// TwinCAT 3 PLC project MoXX_2TilesDemo
// ProgramVersion: 3.1.4026.13
// libraries:
//   Tc2_EtherCAT, * (Beckhoff Automation GmbH)
//   Tc2_MC2, * (Beckhoff Automation GmbH)
//   Tc2_MC2_Camming, * (Beckhoff Automation GmbH)
//   Tc2_NCI, * (Beckhoff Automation GmbH)
//   Tc2_Standard, * (Beckhoff Automation GmbH)
//   Tc2_System, * (Beckhoff Automation GmbH)
//   Tc2_Utilities, * (Beckhoff Automation GmbH)
//   Tc3_Mc3PlanarMotion, * (Beckhoff Automation GmbH)
//   Tc3_Module, * (Beckhoff Automation GmbH)
//   Tc3_Physics, * (Beckhoff Automation GmbH)
//   Tc3_XPlanarStandard, * (Beckhoff Automation GmbH)
//   Tc3_XPlanarUtility, * (Beckhoff Automation GmbH)
// project tree:
//   GVLs/ GVL10_VAR_PRG.TcGVL
//   / PlcTask.TcTTO
//   POUs/10_GeneralPlcBlocks/ Blinker.TcPOU, ClockGenerator.TcPOU, GeneralPlc.TcPOU
//   POUs/10_GeneralPlcBlocks/Components/ FB_Blinker.TcPOU, F_Scaling.TcPOU
//   POUs/CustomerTemplates/GCode/ FB_GCode.TcPOU, I_GCode.TcIO
//   POUs/CustomerTemplates/SwivelMovement/ FB_SwivelMovement.TcPOU, I_SwivelMovement.TcIO
//   POUs/CustomerTemplates/Shake/ FB_ShakeMovement.TcPOU, I_ShakeMovement.TcIO
//   POUs/ FB_MoverApplication.TcPOU, FB_WriteLog.TcPOU, I_MoverApplication.TcIO, MAIN.TcPOU
// real-time tasks:
//   TASK Job Task: cycle default, priority 32
//   TASK MC-Task (MET): cycle T#2ms, priority 3, ADS port 521
//   TASK MC-Task (MPT): cycle T#10ms, priority 8, ADS port 531
//   TASK PlcTask: cycle T#10ms, priority 6, ADS port 352
//   TASK XPlanar Task3: cycle T#250us, priority 1, ADS port 350
// motion (NC):
//   TASK NC-Task 1 SAF: cycle T#2ms, priority 4, ADS port 501
//   TASK NC-Task 1 SVB: cycle T#10ms, priority 9, ADS port 511
//   AXIS MasterShake (id 7)
//     General: UnitFlags=#x00000004
//     OtherSettings: AllowMotionCmdToSlave=true
//     encoder EncType=1
//     drive DrvType=5
//       Analog: TorqueSetpointScale=10, ScaleFactorActTorque=0.1
//       TimeComp: TaskDelayCycles=1
//     controller CtrType=1
//       CtrPara: PriorControlFactor=1
//         Observer: BandWidth=20
//   AXIS Axis a (id 8)
//     OtherSettings: AllowMotionCmdToSlave=true
//     encoder EncType=1
//     drive DrvType=5
//       Analog: TorqueSetpointScale=10, ScaleFactorActTorque=0.1
//       TimeComp: TaskDelayCycles=1
//     controller CtrType=1
//       CtrPara: PriorControlFactor=1
//         Observer: BandWidth=20
//   AXIS Axis b (id 9)
//     OtherSettings: AllowMotionCmdToSlave=true
//     encoder EncType=1
//     drive DrvType=5
//       Analog: TorqueSetpointScale=10, ScaleFactorActTorque=0.1
//       TimeComp: TaskDelayCycles=1
//     controller CtrType=1
//       CtrPara: PriorControlFactor=1
//         Observer: BandWidth=20
//   AXIS Axis x (id 10)
//     OtherSettings: AllowMotionCmdToSlave=true
//     encoder EncType=1
//     drive DrvType=5
//       Analog: TorqueSetpointScale=10, ScaleFactorActTorque=0.1
//       TimeComp: TaskDelayCycles=1
//     controller CtrType=1
//       CtrPara: PriorControlFactor=1
//         Observer: BandWidth=20
//   AXIS Axis y (id 11)
//     OtherSettings: AllowMotionCmdToSlave=true
//     encoder EncType=1
//     drive DrvType=5
//       Analog: TorqueSetpointScale=10, ScaleFactorActTorque=0.1
//       TimeComp: TaskDelayCycles=1
//     controller CtrType=1
//       CtrPara: PriorControlFactor=1
//         Observer: BandWidth=20
//   AXIS Axis 1 (id 1)
//     OtherSettings: AllowMotionCmdToSlave=true
//     encoder EncType=1
//     drive DrvType=5
//       Analog: TorqueSetpointScale=10, ScaleFactorActTorque=0.1
//       TimeComp: TaskDelayCycles=1
//     controller CtrType=1
//       CtrPara: PriorControlFactor=1
//         Observer: BandWidth=20
//   AXIS Axis 2 (id 2)
//     OtherSettings: AllowMotionCmdToSlave=true
//     encoder EncType=1
//     drive DrvType=5
//       Analog: TorqueSetpointScale=10, ScaleFactorActTorque=0.1
//       TimeComp: TaskDelayCycles=1
//     controller CtrType=1
//       CtrPara: PriorControlFactor=1
//         Observer: BandWidth=20
//   AXIS Axis 3 (id 3)
//     OtherSettings: AllowMotionCmdToSlave=true
//     encoder EncType=1
//     drive DrvType=5
//       Analog: TorqueSetpointScale=10, ScaleFactorActTorque=0.1
//       TimeComp: TaskDelayCycles=1
//     controller CtrType=1
//       CtrPara: PriorControlFactor=1
//         Observer: BandWidth=20
//   AXIS Axis 4 (id 4)
//     OtherSettings: AllowMotionCmdToSlave=true
//     encoder EncType=1
//     drive DrvType=5
//       Analog: TorqueSetpointScale=10, ScaleFactorActTorque=0.1
//       TimeComp: TaskDelayCycles=1
//     controller CtrType=1
//       CtrPara: PriorControlFactor=1
//         Observer: BandWidth=20
//   AXIS Axis 5 (id 5)
//     OtherSettings: AllowMotionCmdToSlave=true
//     encoder EncType=1
//     drive DrvType=5
//       Analog: TorqueSetpointScale=10, ScaleFactorActTorque=0.1
//       TimeComp: TaskDelayCycles=1
//     controller CtrType=1
//       CtrPara: PriorControlFactor=1
//         Observer: BandWidth=20
//   AXIS Axis 6 (id 6)
//     OtherSettings: AllowMotionCmdToSlave=true
//     encoder EncType=1
//     drive DrvType=5
//       Analog: TorqueSetpointScale=10, ScaleFactorActTorque=0.1
//       TimeComp: TaskDelayCycles=1
//     controller CtrType=1
//       CtrPara: PriorControlFactor=1
//         Observer: BandWidth=20
// I/O:
//   DEVICE Device 5 (EtherCAT), AmsNetId 5.91.77.10.6.1
//     Term 1 (APS4322-7000) [APS4322-7000 Drive]
//       Term 2 (APS4322-5000) [APS4322-5000 Feedback]
//     Term 3 (APS4322-7000) [APS4322-7000 Drive]
//       Term 4 (APS4322-5000) [APS4322-5000 Feedback]
//   DEVICE Gerät 4 (EtherCAT), AmsNetId 169.254.59.222.5.1
//     Box 5 (EP2316-0003) [EP2316-0003 8 K. Dig. Ein, 10µs, 8 K. Dig. Aus 24V, 0,5A, Diagnose, 10-Pol Steckverbinder]
// variable links:
//   Device 5 (EtherCAT) <-> TcCOM Objects/XPlanar/Part1/Tile1
//     Term 1 (APS4322-7000)/APS Comm Inputs/CommStatusWord <-> Data Pointer/MoverCommStatusWord
//     Term 1 (APS4322-7000)/APS Comm Inputs/Data {1..4} <-> Data Pointer/MoverCommDataIn[{0..3}]  (4 links)
//     Term 1 (APS4322-7000)/APS Comm Outputs/CommControlWord <-> Data Pointer/MoverCommControlWord
//     Term 1 (APS4322-7000)/APS Comm Outputs/Data 1 <-> Data Pointer/MoverCommDataOut
//     Term 1 (APS4322-7000)/APS Diagdata/DC Link Voltage <-> Data Pointer/DcLinkVoltage
//     Term 1 (APS4322-7000)/APS Diagdata/Power supply current <-> Data Pointer/PowerSupplyCurrent
//     Term 1 (APS4322-7000)/APS Inputs/StatusWord <-> Data Pointer/PowerUnitStatusWord
//     Term 1 (APS4322-7000)/APS Outputs/ControlWord <-> Data Pointer/PowerUnitControlWord
//     Term 1 (APS4322-7000)/APS Outputs/Current D 0X0 <-> Data Pointer/DCurrentSetPoints[0]
//     Term 1 (APS4322-7000)/APS Outputs/Current D 0X1 <-> Data Pointer/DCurrentSetPoints[1]
//     Term 1 (APS4322-7000)/APS Outputs/Current D 0X2 <-> Data Pointer/DCurrentSetPoints[2]
//     Term 1 (APS4322-7000)/APS Outputs/Current D 1X0 <-> Data Pointer/DCurrentSetPoints[6]
//     Term 1 (APS4322-7000)/APS Outputs/Current D 1X1 <-> Data Pointer/DCurrentSetPoints[7]
//     Term 1 (APS4322-7000)/APS Outputs/Current D 1X2 <-> Data Pointer/DCurrentSetPoints[8]
//     Term 1 (APS4322-7000)/APS Outputs/Current D 2X0 <-> Data Pointer/DCurrentSetPoints[12]
//     Term 1 (APS4322-7000)/APS Outputs/Current D 2X1 <-> Data Pointer/DCurrentSetPoints[13]
//     Term 1 (APS4322-7000)/APS Outputs/Current D 2X2 <-> Data Pointer/DCurrentSetPoints[14]
//     Term 1 (APS4322-7000)/APS Outputs/Current D 3X0 <-> Data Pointer/DCurrentSetPoints[18]
//     Term 1 (APS4322-7000)/APS Outputs/Current D 3X1 <-> Data Pointer/DCurrentSetPoints[19]
//     Term 1 (APS4322-7000)/APS Outputs/Current D 3X2 <-> Data Pointer/DCurrentSetPoints[20]
//     Term 1 (APS4322-7000)/APS Outputs/Current D 0Y0 <-> Data Pointer/DCurrentSetPoints[3]
//     Term 1 (APS4322-7000)/APS Outputs/Current D 0Y1 <-> Data Pointer/DCurrentSetPoints[4]
//     Term 1 (APS4322-7000)/APS Outputs/Current D 0Y2 <-> Data Pointer/DCurrentSetPoints[5]
//     Term 1 (APS4322-7000)/APS Outputs/Current D 1Y0 <-> Data Pointer/DCurrentSetPoints[9]
//     Term 1 (APS4322-7000)/APS Outputs/Current D 1Y1 <-> Data Pointer/DCurrentSetPoints[10]
//     Term 1 (APS4322-7000)/APS Outputs/Current D 1Y2 <-> Data Pointer/DCurrentSetPoints[11]
//     Term 1 (APS4322-7000)/APS Outputs/Current D 2Y0 <-> Data Pointer/DCurrentSetPoints[15]
//     Term 1 (APS4322-7000)/APS Outputs/Current D 2Y1 <-> Data Pointer/DCurrentSetPoints[16]
//     Term 1 (APS4322-7000)/APS Outputs/Current D 2Y2 <-> Data Pointer/DCurrentSetPoints[17]
//     Term 1 (APS4322-7000)/APS Outputs/Current D 3Y0 <-> Data Pointer/DCurrentSetPoints[21]
//     Term 1 (APS4322-7000)/APS Outputs/Current D 3Y1 <-> Data Pointer/DCurrentSetPoints[22]
//     Term 1 (APS4322-7000)/APS Outputs/Current D 3Y2 <-> Data Pointer/DCurrentSetPoints[23]
//     Term 1 (APS4322-7000)/APS Outputs/Current Q 0X0 <-> Data Pointer/QCurrentSetPoints[0]
//     Term 1 (APS4322-7000)/APS Outputs/Current Q 0X1 <-> Data Pointer/QCurrentSetPoints[1]
//     Term 1 (APS4322-7000)/APS Outputs/Current Q 0X2 <-> Data Pointer/QCurrentSetPoints[2]
//     Term 1 (APS4322-7000)/APS Outputs/Current Q 1X0 <-> Data Pointer/QCurrentSetPoints[6]
//     Term 1 (APS4322-7000)/APS Outputs/Current Q 1X1 <-> Data Pointer/QCurrentSetPoints[7]
//     Term 1 (APS4322-7000)/APS Outputs/Current Q 1X2 <-> Data Pointer/QCurrentSetPoints[8]
//     Term 1 (APS4322-7000)/APS Outputs/Current Q 2X0 <-> Data Pointer/QCurrentSetPoints[12]
//     Term 1 (APS4322-7000)/APS Outputs/Current Q 2X1 <-> Data Pointer/QCurrentSetPoints[13]
//     Term 1 (APS4322-7000)/APS Outputs/Current Q 2X2 <-> Data Pointer/QCurrentSetPoints[14]
//     Term 1 (APS4322-7000)/APS Outputs/Current Q 3X0 <-> Data Pointer/QCurrentSetPoints[18]
//     Term 1 (APS4322-7000)/APS Outputs/Current Q 3X1 <-> Data Pointer/QCurrentSetPoints[19]
//     Term 1 (APS4322-7000)/APS Outputs/Current Q 3X2 <-> Data Pointer/QCurrentSetPoints[20]
//     Term 1 (APS4322-7000)/APS Outputs/Current Q 0Y0 <-> Data Pointer/QCurrentSetPoints[3]
//     Term 1 (APS4322-7000)/APS Outputs/Current Q 0Y1 <-> Data Pointer/QCurrentSetPoints[4]
//     Term 1 (APS4322-7000)/APS Outputs/Current Q 0Y2 <-> Data Pointer/QCurrentSetPoints[5]
//     Term 1 (APS4322-7000)/APS Outputs/Current Q 1Y0 <-> Data Pointer/QCurrentSetPoints[9]
//     Term 1 (APS4322-7000)/APS Outputs/Current Q 1Y1 <-> Data Pointer/QCurrentSetPoints[10]
//     Term 1 (APS4322-7000)/APS Outputs/Current Q 1Y2 <-> Data Pointer/QCurrentSetPoints[11]
//     Term 1 (APS4322-7000)/APS Outputs/Current Q 2Y0 <-> Data Pointer/QCurrentSetPoints[15]
//     Term 1 (APS4322-7000)/APS Outputs/Current Q 2Y1 <-> Data Pointer/QCurrentSetPoints[16]
//     Term 1 (APS4322-7000)/APS Outputs/Current Q 2Y2 <-> Data Pointer/QCurrentSetPoints[17]
//     Term 1 (APS4322-7000)/APS Outputs/Current Q 3Y0 <-> Data Pointer/QCurrentSetPoints[21]
//     Term 1 (APS4322-7000)/APS Outputs/Current Q 3Y1 <-> Data Pointer/QCurrentSetPoints[22]
//     Term 1 (APS4322-7000)/APS Outputs/Current Q 3Y2 <-> Data Pointer/QCurrentSetPoints[23]
//     Term 1 (APS4322-7000)/APS Outputs/PhiE 0X0 <-> Data Pointer/PhiSetPoints[0]
//     Term 1 (APS4322-7000)/APS Outputs/PhiE 0X1 <-> Data Pointer/PhiSetPoints[1]
//     Term 1 (APS4322-7000)/APS Outputs/PhiE 0X2 <-> Data Pointer/PhiSetPoints[2]
//     Term 1 (APS4322-7000)/APS Outputs/PhiE 1X0 <-> Data Pointer/PhiSetPoints[6]
//     Term 1 (APS4322-7000)/APS Outputs/PhiE 1X1 <-> Data Pointer/PhiSetPoints[7]
//     Term 1 (APS4322-7000)/APS Outputs/PhiE 1X2 <-> Data Pointer/PhiSetPoints[8]
//     Term 1 (APS4322-7000)/APS Outputs/PhiE 2X0 <-> Data Pointer/PhiSetPoints[12]
//     Term 1 (APS4322-7000)/APS Outputs/PhiE 2X1 <-> Data Pointer/PhiSetPoints[13]
//     Term 1 (APS4322-7000)/APS Outputs/PhiE 2X2 <-> Data Pointer/PhiSetPoints[14]
//     Term 1 (APS4322-7000)/APS Outputs/PhiE 3X0 <-> Data Pointer/PhiSetPoints[18]
//     Term 1 (APS4322-7000)/APS Outputs/PhiE 3X1 <-> Data Pointer/PhiSetPoints[19]
//     Term 1 (APS4322-7000)/APS Outputs/PhiE 3X2 <-> Data Pointer/PhiSetPoints[20]
//     Term 1 (APS4322-7000)/APS Outputs/PhiE 0Y0 <-> Data Pointer/PhiSetPoints[3]
//     Term 1 (APS4322-7000)/APS Outputs/PhiE 0Y1 <-> Data Pointer/PhiSetPoints[4]
//     Term 1 (APS4322-7000)/APS Outputs/PhiE 0Y2 <-> Data Pointer/PhiSetPoints[5]
//     Term 1 (APS4322-7000)/APS Outputs/PhiE 1Y0 <-> Data Pointer/PhiSetPoints[9]
//     Term 1 (APS4322-7000)/APS Outputs/PhiE 1Y1 <-> Data Pointer/PhiSetPoints[10]
//     Term 1 (APS4322-7000)/APS Outputs/PhiE 1Y2 <-> Data Pointer/PhiSetPoints[11]
//     Term 1 (APS4322-7000)/APS Outputs/PhiE 2Y0 <-> Data Pointer/PhiSetPoints[15]
//     Term 1 (APS4322-7000)/APS Outputs/PhiE 2Y1 <-> Data Pointer/PhiSetPoints[16]
//     Term 1 (APS4322-7000)/APS Outputs/PhiE 2Y2 <-> Data Pointer/PhiSetPoints[17]
//     Term 1 (APS4322-7000)/APS Outputs/PhiE 3Y0 <-> Data Pointer/PhiSetPoints[21]
//     Term 1 (APS4322-7000)/APS Outputs/PhiE 3Y1 <-> Data Pointer/PhiSetPoints[22]
//     Term 1 (APS4322-7000)/APS Outputs/PhiE 3Y2 <-> Data Pointer/PhiSetPoints[23]
//     Term 1 (APS4322-7000)/Term 2 (APS4322-5000)/FB Inputs/A{0..8 step 2} X-Field <-> Data Pointer/HallSensorFieldsXYZ[{0..12 step 3}]  (5 links)
//     Term 1 (APS4322-7000)/Term 2 (APS4322-5000)/FB Inputs/A{0..8 step 2} Y-Field <-> Data Pointer/HallSensorFieldsXYZ[{1..13 step 3}]  (5 links)
//     Term 1 (APS4322-7000)/Term 2 (APS4322-5000)/FB Inputs/A{0..8 step 2} Z-Field <-> Data Pointer/HallSensorFieldsXYZ[{2..14 step 3}]  (5 links)
//     Term 1 (APS4322-7000)/Term 2 (APS4322-5000)/FB Inputs/B{1..9 step 2} X-Field <-> Data Pointer/HallSensorFieldsXYZ[{15..27 step 3}]  (5 links)
//     Term 1 (APS4322-7000)/Term 2 (APS4322-5000)/FB Inputs/B{1..9 step 2} Y-Field <-> Data Pointer/HallSensorFieldsXYZ[{16..28 step 3}]  (5 links)
//     Term 1 (APS4322-7000)/Term 2 (APS4322-5000)/FB Inputs/B{1..9 step 2} Z-Field <-> Data Pointer/HallSensorFieldsXYZ[{17..29 step 3}]  (5 links)
//     Term 1 (APS4322-7000)/Term 2 (APS4322-5000)/FB Inputs/C{0..8 step 2} X-Field <-> Data Pointer/HallSensorFieldsXYZ[{30..42 step 3}]  (5 links)
//     Term 1 (APS4322-7000)/Term 2 (APS4322-5000)/FB Inputs/C{0..8 step 2} Y-Field <-> Data Pointer/HallSensorFieldsXYZ[{31..43 step 3}]  (5 links)
//     Term 1 (APS4322-7000)/Term 2 (APS4322-5000)/FB Inputs/C{0..8 step 2} Z-Field <-> Data Pointer/HallSensorFieldsXYZ[{32..44 step 3}]  (5 links)
//     Term 1 (APS4322-7000)/Term 2 (APS4322-5000)/FB Inputs/D{1..9 step 2} X-Field <-> Data Pointer/HallSensorFieldsXYZ[{45..57 step 3}]  (5 links)
//     Term 1 (APS4322-7000)/Term 2 (APS4322-5000)/FB Inputs/D{1..9 step 2} Y-Field <-> Data Pointer/HallSensorFieldsXYZ[{46..58 step 3}]  (5 links)
//     Term 1 (APS4322-7000)/Term 2 (APS4322-5000)/FB Inputs/D{1..9 step 2} Z-Field <-> Data Pointer/HallSensorFieldsXYZ[{47..59 step 3}]  (5 links)
//     Term 1 (APS4322-7000)/Term 2 (APS4322-5000)/FB Inputs/E{0..8 step 2} X-Field <-> Data Pointer/HallSensorFieldsXYZ[{60..72 step 3}]  (5 links)
//     Term 1 (APS4322-7000)/Term 2 (APS4322-5000)/FB Inputs/E{0..8 step 2} Y-Field <-> Data Pointer/HallSensorFieldsXYZ[{61..73 step 3}]  (5 links)
//     Term 1 (APS4322-7000)/Term 2 (APS4322-5000)/FB Inputs/E{0..8 step 2} Z-Field <-> Data Pointer/HallSensorFieldsXYZ[{62..74 step 3}]  (5 links)
//     Term 1 (APS4322-7000)/Term 2 (APS4322-5000)/FB Inputs/F{1..9 step 2} X-Field <-> Data Pointer/HallSensorFieldsXYZ[{75..87 step 3}]  (5 links)
//     Term 1 (APS4322-7000)/Term 2 (APS4322-5000)/FB Inputs/F{1..9 step 2} Y-Field <-> Data Pointer/HallSensorFieldsXYZ[{76..88 step 3}]  (5 links)
//     Term 1 (APS4322-7000)/Term 2 (APS4322-5000)/FB Inputs/F{1..9 step 2} Z-Field <-> Data Pointer/HallSensorFieldsXYZ[{77..89 step 3}]  (5 links)
//     Term 1 (APS4322-7000)/Term 2 (APS4322-5000)/FB Inputs/G{0..8 step 2} X-Field <-> Data Pointer/HallSensorFieldsXYZ[{90..102 step 3}]  (5 links)
//     Term 1 (APS4322-7000)/Term 2 (APS4322-5000)/FB Inputs/G{0..8 step 2} Y-Field <-> Data Pointer/HallSensorFieldsXYZ[{91..103 step 3}]  (5 links)
//     Term 1 (APS4322-7000)/Term 2 (APS4322-5000)/FB Inputs/G{0..8 step 2} Z-Field <-> Data Pointer/HallSensorFieldsXYZ[{92..104 step 3}]  (5 links)
//     Term 1 (APS4322-7000)/Term 2 (APS4322-5000)/FB Inputs/H{1..9 step 2} X-Field <-> Data Pointer/HallSensorFieldsXYZ[{105..117 step 3}]  (5 links)
//     Term 1 (APS4322-7000)/Term 2 (APS4322-5000)/FB Inputs/H{1..9 step 2} Y-Field <-> Data Pointer/HallSensorFieldsXYZ[{106..118 step 3}]  (5 links)
//     Term 1 (APS4322-7000)/Term 2 (APS4322-5000)/FB Inputs/H{1..9 step 2} Z-Field <-> Data Pointer/HallSensorFieldsXYZ[{107..119 step 3}]  (5 links)
//     Term 1 (APS4322-7000)/Term 2 (APS4322-5000)/FB Inputs/I{0..8 step 2} X-Field <-> Data Pointer/HallSensorFieldsXYZ[{120..132 step 3}]  (5 links)
//     Term 1 (APS4322-7000)/Term 2 (APS4322-5000)/FB Inputs/I{0..8 step 2} Y-Field <-> Data Pointer/HallSensorFieldsXYZ[{121..133 step 3}]  (5 links)
//     Term 1 (APS4322-7000)/Term 2 (APS4322-5000)/FB Inputs/I{0..8 step 2} Z-Field <-> Data Pointer/HallSensorFieldsXYZ[{122..134 step 3}]  (5 links)
//     Term 1 (APS4322-7000)/Term 2 (APS4322-5000)/FB Inputs/J{1..9 step 2} X-Field <-> Data Pointer/HallSensorFieldsXYZ[{135..147 step 3}]  (5 links)
//     Term 1 (APS4322-7000)/Term 2 (APS4322-5000)/FB Inputs/J{1..9 step 2} Y-Field <-> Data Pointer/HallSensorFieldsXYZ[{136..148 step 3}]  (5 links)
//     Term 1 (APS4322-7000)/Term 2 (APS4322-5000)/FB Inputs/J{1..9 step 2} Z-Field <-> Data Pointer/HallSensorFieldsXYZ[{137..149 step 3}]  (5 links)
//     Term 1 (APS4322-7000)/Term 2 (APS4322-5000)/FB Inputs/Status <-> Data Pointer/FeedbackStatus
//   Device 5 (EtherCAT) <-> TcCOM Objects/XPlanar/Part1/Tile2
//     Term 3 (APS4322-7000)/APS Comm Inputs/CommStatusWord <-> Data Pointer/MoverCommStatusWord
//     Term 3 (APS4322-7000)/APS Comm Inputs/Data {1..4} <-> Data Pointer/MoverCommDataIn[{0..3}]  (4 links)
//     Term 3 (APS4322-7000)/APS Comm Outputs/CommControlWord <-> Data Pointer/MoverCommControlWord
//     Term 3 (APS4322-7000)/APS Comm Outputs/Data 1 <-> Data Pointer/MoverCommDataOut
//     Term 3 (APS4322-7000)/APS Diagdata/DC Link Voltage <-> Data Pointer/DcLinkVoltage
//     Term 3 (APS4322-7000)/APS Diagdata/Power supply current <-> Data Pointer/PowerSupplyCurrent
//     Term 3 (APS4322-7000)/APS Inputs/StatusWord <-> Data Pointer/PowerUnitStatusWord
//     Term 3 (APS4322-7000)/APS Outputs/ControlWord <-> Data Pointer/PowerUnitControlWord
//     Term 3 (APS4322-7000)/APS Outputs/Current D 0X0 <-> Data Pointer/DCurrentSetPoints[0]
//     Term 3 (APS4322-7000)/APS Outputs/Current D 0X1 <-> Data Pointer/DCurrentSetPoints[1]
//     Term 3 (APS4322-7000)/APS Outputs/Current D 0X2 <-> Data Pointer/DCurrentSetPoints[2]
//     Term 3 (APS4322-7000)/APS Outputs/Current D 1X0 <-> Data Pointer/DCurrentSetPoints[6]
//     Term 3 (APS4322-7000)/APS Outputs/Current D 1X1 <-> Data Pointer/DCurrentSetPoints[7]
//     Term 3 (APS4322-7000)/APS Outputs/Current D 1X2 <-> Data Pointer/DCurrentSetPoints[8]
//     Term 3 (APS4322-7000)/APS Outputs/Current D 2X0 <-> Data Pointer/DCurrentSetPoints[12]
//     Term 3 (APS4322-7000)/APS Outputs/Current D 2X1 <-> Data Pointer/DCurrentSetPoints[13]
//     Term 3 (APS4322-7000)/APS Outputs/Current D 2X2 <-> Data Pointer/DCurrentSetPoints[14]
//     Term 3 (APS4322-7000)/APS Outputs/Current D 3X0 <-> Data Pointer/DCurrentSetPoints[18]
//     Term 3 (APS4322-7000)/APS Outputs/Current D 3X1 <-> Data Pointer/DCurrentSetPoints[19]
//     Term 3 (APS4322-7000)/APS Outputs/Current D 3X2 <-> Data Pointer/DCurrentSetPoints[20]
//     Term 3 (APS4322-7000)/APS Outputs/Current D 0Y0 <-> Data Pointer/DCurrentSetPoints[3]
//     Term 3 (APS4322-7000)/APS Outputs/Current D 0Y1 <-> Data Pointer/DCurrentSetPoints[4]
//     Term 3 (APS4322-7000)/APS Outputs/Current D 0Y2 <-> Data Pointer/DCurrentSetPoints[5]
//     Term 3 (APS4322-7000)/APS Outputs/Current D 1Y0 <-> Data Pointer/DCurrentSetPoints[9]
//     Term 3 (APS4322-7000)/APS Outputs/Current D 1Y1 <-> Data Pointer/DCurrentSetPoints[10]
//     Term 3 (APS4322-7000)/APS Outputs/Current D 1Y2 <-> Data Pointer/DCurrentSetPoints[11]
//     Term 3 (APS4322-7000)/APS Outputs/Current D 2Y0 <-> Data Pointer/DCurrentSetPoints[15]
//     Term 3 (APS4322-7000)/APS Outputs/Current D 2Y1 <-> Data Pointer/DCurrentSetPoints[16]
//     Term 3 (APS4322-7000)/APS Outputs/Current D 2Y2 <-> Data Pointer/DCurrentSetPoints[17]
//     Term 3 (APS4322-7000)/APS Outputs/Current D 3Y0 <-> Data Pointer/DCurrentSetPoints[21]
//     Term 3 (APS4322-7000)/APS Outputs/Current D 3Y1 <-> Data Pointer/DCurrentSetPoints[22]
//     Term 3 (APS4322-7000)/APS Outputs/Current D 3Y2 <-> Data Pointer/DCurrentSetPoints[23]
//     Term 3 (APS4322-7000)/APS Outputs/Current Q 0X0 <-> Data Pointer/QCurrentSetPoints[0]
//     Term 3 (APS4322-7000)/APS Outputs/Current Q 0X1 <-> Data Pointer/QCurrentSetPoints[1]
//     Term 3 (APS4322-7000)/APS Outputs/Current Q 0X2 <-> Data Pointer/QCurrentSetPoints[2]
//     Term 3 (APS4322-7000)/APS Outputs/Current Q 1X0 <-> Data Pointer/QCurrentSetPoints[6]
//     Term 3 (APS4322-7000)/APS Outputs/Current Q 1X1 <-> Data Pointer/QCurrentSetPoints[7]
//     Term 3 (APS4322-7000)/APS Outputs/Current Q 1X2 <-> Data Pointer/QCurrentSetPoints[8]
//     Term 3 (APS4322-7000)/APS Outputs/Current Q 2X0 <-> Data Pointer/QCurrentSetPoints[12]
//     Term 3 (APS4322-7000)/APS Outputs/Current Q 2X1 <-> Data Pointer/QCurrentSetPoints[13]
//     Term 3 (APS4322-7000)/APS Outputs/Current Q 2X2 <-> Data Pointer/QCurrentSetPoints[14]
//     Term 3 (APS4322-7000)/APS Outputs/Current Q 3X0 <-> Data Pointer/QCurrentSetPoints[18]
//     Term 3 (APS4322-7000)/APS Outputs/Current Q 3X1 <-> Data Pointer/QCurrentSetPoints[19]
//     Term 3 (APS4322-7000)/APS Outputs/Current Q 3X2 <-> Data Pointer/QCurrentSetPoints[20]
//     Term 3 (APS4322-7000)/APS Outputs/Current Q 0Y0 <-> Data Pointer/QCurrentSetPoints[3]
//     Term 3 (APS4322-7000)/APS Outputs/Current Q 0Y1 <-> Data Pointer/QCurrentSetPoints[4]
//     Term 3 (APS4322-7000)/APS Outputs/Current Q 0Y2 <-> Data Pointer/QCurrentSetPoints[5]
//     Term 3 (APS4322-7000)/APS Outputs/Current Q 1Y0 <-> Data Pointer/QCurrentSetPoints[9]
//     Term 3 (APS4322-7000)/APS Outputs/Current Q 1Y1 <-> Data Pointer/QCurrentSetPoints[10]
//     Term 3 (APS4322-7000)/APS Outputs/Current Q 1Y2 <-> Data Pointer/QCurrentSetPoints[11]
//     Term 3 (APS4322-7000)/APS Outputs/Current Q 2Y0 <-> Data Pointer/QCurrentSetPoints[15]
//     Term 3 (APS4322-7000)/APS Outputs/Current Q 2Y1 <-> Data Pointer/QCurrentSetPoints[16]
//     Term 3 (APS4322-7000)/APS Outputs/Current Q 2Y2 <-> Data Pointer/QCurrentSetPoints[17]
//     Term 3 (APS4322-7000)/APS Outputs/Current Q 3Y0 <-> Data Pointer/QCurrentSetPoints[21]
//     Term 3 (APS4322-7000)/APS Outputs/Current Q 3Y1 <-> Data Pointer/QCurrentSetPoints[22]
//     Term 3 (APS4322-7000)/APS Outputs/Current Q 3Y2 <-> Data Pointer/QCurrentSetPoints[23]
//     Term 3 (APS4322-7000)/APS Outputs/PhiE 0X0 <-> Data Pointer/PhiSetPoints[0]
//     Term 3 (APS4322-7000)/APS Outputs/PhiE 0X1 <-> Data Pointer/PhiSetPoints[1]
//     Term 3 (APS4322-7000)/APS Outputs/PhiE 0X2 <-> Data Pointer/PhiSetPoints[2]
//     Term 3 (APS4322-7000)/APS Outputs/PhiE 1X0 <-> Data Pointer/PhiSetPoints[6]
//     Term 3 (APS4322-7000)/APS Outputs/PhiE 1X1 <-> Data Pointer/PhiSetPoints[7]
//     Term 3 (APS4322-7000)/APS Outputs/PhiE 1X2 <-> Data Pointer/PhiSetPoints[8]
//     Term 3 (APS4322-7000)/APS Outputs/PhiE 2X0 <-> Data Pointer/PhiSetPoints[12]
//     Term 3 (APS4322-7000)/APS Outputs/PhiE 2X1 <-> Data Pointer/PhiSetPoints[13]
//     Term 3 (APS4322-7000)/APS Outputs/PhiE 2X2 <-> Data Pointer/PhiSetPoints[14]
//     Term 3 (APS4322-7000)/APS Outputs/PhiE 3X0 <-> Data Pointer/PhiSetPoints[18]
//     Term 3 (APS4322-7000)/APS Outputs/PhiE 3X1 <-> Data Pointer/PhiSetPoints[19]
//     Term 3 (APS4322-7000)/APS Outputs/PhiE 3X2 <-> Data Pointer/PhiSetPoints[20]
//     Term 3 (APS4322-7000)/APS Outputs/PhiE 0Y0 <-> Data Pointer/PhiSetPoints[3]
//     Term 3 (APS4322-7000)/APS Outputs/PhiE 0Y1 <-> Data Pointer/PhiSetPoints[4]
//     Term 3 (APS4322-7000)/APS Outputs/PhiE 0Y2 <-> Data Pointer/PhiSetPoints[5]
//     Term 3 (APS4322-7000)/APS Outputs/PhiE 1Y0 <-> Data Pointer/PhiSetPoints[9]
//     Term 3 (APS4322-7000)/APS Outputs/PhiE 1Y1 <-> Data Pointer/PhiSetPoints[10]
//     Term 3 (APS4322-7000)/APS Outputs/PhiE 1Y2 <-> Data Pointer/PhiSetPoints[11]
//     Term 3 (APS4322-7000)/APS Outputs/PhiE 2Y0 <-> Data Pointer/PhiSetPoints[15]
//     Term 3 (APS4322-7000)/APS Outputs/PhiE 2Y1 <-> Data Pointer/PhiSetPoints[16]
//     Term 3 (APS4322-7000)/APS Outputs/PhiE 2Y2 <-> Data Pointer/PhiSetPoints[17]
//     Term 3 (APS4322-7000)/APS Outputs/PhiE 3Y0 <-> Data Pointer/PhiSetPoints[21]
//     Term 3 (APS4322-7000)/APS Outputs/PhiE 3Y1 <-> Data Pointer/PhiSetPoints[22]
//     Term 3 (APS4322-7000)/APS Outputs/PhiE 3Y2 <-> Data Pointer/PhiSetPoints[23]
//     Term 3 (APS4322-7000)/Term 4 (APS4322-5000)/FB Inputs/A{0..8 step 2} X-Field <-> Data Pointer/HallSensorFieldsXYZ[{0..12 step 3}]  (5 links)
//     Term 3 (APS4322-7000)/Term 4 (APS4322-5000)/FB Inputs/A{0..8 step 2} Y-Field <-> Data Pointer/HallSensorFieldsXYZ[{1..13 step 3}]  (5 links)
//     Term 3 (APS4322-7000)/Term 4 (APS4322-5000)/FB Inputs/A{0..8 step 2} Z-Field <-> Data Pointer/HallSensorFieldsXYZ[{2..14 step 3}]  (5 links)
//     Term 3 (APS4322-7000)/Term 4 (APS4322-5000)/FB Inputs/B{1..9 step 2} X-Field <-> Data Pointer/HallSensorFieldsXYZ[{15..27 step 3}]  (5 links)
//     Term 3 (APS4322-7000)/Term 4 (APS4322-5000)/FB Inputs/B{1..9 step 2} Y-Field <-> Data Pointer/HallSensorFieldsXYZ[{16..28 step 3}]  (5 links)
//     Term 3 (APS4322-7000)/Term 4 (APS4322-5000)/FB Inputs/B{1..9 step 2} Z-Field <-> Data Pointer/HallSensorFieldsXYZ[{17..29 step 3}]  (5 links)
//     Term 3 (APS4322-7000)/Term 4 (APS4322-5000)/FB Inputs/C{0..8 step 2} X-Field <-> Data Pointer/HallSensorFieldsXYZ[{30..42 step 3}]  (5 links)
//     Term 3 (APS4322-7000)/Term 4 (APS4322-5000)/FB Inputs/C{0..8 step 2} Y-Field <-> Data Pointer/HallSensorFieldsXYZ[{31..43 step 3}]  (5 links)
//     Term 3 (APS4322-7000)/Term 4 (APS4322-5000)/FB Inputs/C{0..8 step 2} Z-Field <-> Data Pointer/HallSensorFieldsXYZ[{32..44 step 3}]  (5 links)
//     Term 3 (APS4322-7000)/Term 4 (APS4322-5000)/FB Inputs/D{1..9 step 2} X-Field <-> Data Pointer/HallSensorFieldsXYZ[{45..57 step 3}]  (5 links)
//     Term 3 (APS4322-7000)/Term 4 (APS4322-5000)/FB Inputs/D{1..9 step 2} Y-Field <-> Data Pointer/HallSensorFieldsXYZ[{46..58 step 3}]  (5 links)
//     Term 3 (APS4322-7000)/Term 4 (APS4322-5000)/FB Inputs/D{1..9 step 2} Z-Field <-> Data Pointer/HallSensorFieldsXYZ[{47..59 step 3}]  (5 links)
//     Term 3 (APS4322-7000)/Term 4 (APS4322-5000)/FB Inputs/E{0..8 step 2} X-Field <-> Data Pointer/HallSensorFieldsXYZ[{60..72 step 3}]  (5 links)
//     Term 3 (APS4322-7000)/Term 4 (APS4322-5000)/FB Inputs/E{0..8 step 2} Y-Field <-> Data Pointer/HallSensorFieldsXYZ[{61..73 step 3}]  (5 links)
//     Term 3 (APS4322-7000)/Term 4 (APS4322-5000)/FB Inputs/E{0..8 step 2} Z-Field <-> Data Pointer/HallSensorFieldsXYZ[{62..74 step 3}]  (5 links)
//     Term 3 (APS4322-7000)/Term 4 (APS4322-5000)/FB Inputs/F{1..9 step 2} X-Field <-> Data Pointer/HallSensorFieldsXYZ[{75..87 step 3}]  (5 links)
//     Term 3 (APS4322-7000)/Term 4 (APS4322-5000)/FB Inputs/F{1..9 step 2} Y-Field <-> Data Pointer/HallSensorFieldsXYZ[{76..88 step 3}]  (5 links)
//     Term 3 (APS4322-7000)/Term 4 (APS4322-5000)/FB Inputs/F{1..9 step 2} Z-Field <-> Data Pointer/HallSensorFieldsXYZ[{77..89 step 3}]  (5 links)
//     Term 3 (APS4322-7000)/Term 4 (APS4322-5000)/FB Inputs/G{0..8 step 2} X-Field <-> Data Pointer/HallSensorFieldsXYZ[{90..102 step 3}]  (5 links)
//     Term 3 (APS4322-7000)/Term 4 (APS4322-5000)/FB Inputs/G{0..8 step 2} Y-Field <-> Data Pointer/HallSensorFieldsXYZ[{91..103 step 3}]  (5 links)
//     Term 3 (APS4322-7000)/Term 4 (APS4322-5000)/FB Inputs/G{0..8 step 2} Z-Field <-> Data Pointer/HallSensorFieldsXYZ[{92..104 step 3}]  (5 links)
//     Term 3 (APS4322-7000)/Term 4 (APS4322-5000)/FB Inputs/H{1..9 step 2} X-Field <-> Data Pointer/HallSensorFieldsXYZ[{105..117 step 3}]  (5 links)
//     Term 3 (APS4322-7000)/Term 4 (APS4322-5000)/FB Inputs/H{1..9 step 2} Y-Field <-> Data Pointer/HallSensorFieldsXYZ[{106..118 step 3}]  (5 links)
//     Term 3 (APS4322-7000)/Term 4 (APS4322-5000)/FB Inputs/H{1..9 step 2} Z-Field <-> Data Pointer/HallSensorFieldsXYZ[{107..119 step 3}]  (5 links)
//     Term 3 (APS4322-7000)/Term 4 (APS4322-5000)/FB Inputs/I{0..8 step 2} X-Field <-> Data Pointer/HallSensorFieldsXYZ[{120..132 step 3}]  (5 links)
//     Term 3 (APS4322-7000)/Term 4 (APS4322-5000)/FB Inputs/I{0..8 step 2} Y-Field <-> Data Pointer/HallSensorFieldsXYZ[{121..133 step 3}]  (5 links)
//     Term 3 (APS4322-7000)/Term 4 (APS4322-5000)/FB Inputs/I{0..8 step 2} Z-Field <-> Data Pointer/HallSensorFieldsXYZ[{122..134 step 3}]  (5 links)
//     Term 3 (APS4322-7000)/Term 4 (APS4322-5000)/FB Inputs/J{1..9 step 2} X-Field <-> Data Pointer/HallSensorFieldsXYZ[{135..147 step 3}]  (5 links)
//     Term 3 (APS4322-7000)/Term 4 (APS4322-5000)/FB Inputs/J{1..9 step 2} Y-Field <-> Data Pointer/HallSensorFieldsXYZ[{136..148 step 3}]  (5 links)
//     Term 3 (APS4322-7000)/Term 4 (APS4322-5000)/FB Inputs/J{1..9 step 2} Z-Field <-> Data Pointer/HallSensorFieldsXYZ[{137..149 step 3}]  (5 links)
//     Term 3 (APS4322-7000)/Term 4 (APS4322-5000)/FB Inputs/Status <-> Data Pointer/FeedbackStatus
//   XPlanar MC Project/Axes/Mover4220_1 <-> TcCOM Objects/XPlanar/Mover4220_1
//     IoToMc/STD <-> OutputsToNC3/HWToNC3
//     McToIo/STD <-> InputsFromNC3/NC3ToHW
//   XPlanar MC Project/Axes/Mover4220_2 <-> TcCOM Objects/XPlanar/Mover4220_2
//     IoToMc/STD <-> OutputsToNC3/HWToNC3
//     McToIo/STD <-> InputsFromNC3/NC3ToHW
//   (this object) <-> Device 4 (EtherCAT)/Box 5 (EP2316-0003)
//     PlcTask Inputs/MAIN.IbSwitch <-> DIG Inputs/Input 3
//     PlcTask Inputs/MAIN.IbSwitchRestart <-> DIG Inputs/Input 4
//   (this object) <-> NC-Task 1 SAF/Axes/Axis 1
//     PlcTask Inputs/MAIN.mover[1].fbSwivelMovement.stAxisMaster.NcToPlc <-> Outputs/ToPlc
//     PlcTask Outputs/MAIN.mover[1].fbSwivelMovement.stAxisMaster.PlcToNc <-> Inputs/FromPlc
//   (this object) <-> NC-Task 1 SAF/Axes/Axis 2
//     PlcTask Inputs/MAIN.mover[1].fbSwivelMovement.stAxisX.NcToPlc <-> Outputs/ToPlc
//     PlcTask Outputs/MAIN.mover[1].fbSwivelMovement.stAxisX.PlcToNc <-> Inputs/FromPlc
//   (this object) <-> NC-Task 1 SAF/Axes/Axis 3
//     PlcTask Inputs/MAIN.mover[1].fbSwivelMovement.stAxisY.NcToPlc <-> Outputs/ToPlc
//     PlcTask Outputs/MAIN.mover[1].fbSwivelMovement.stAxisY.PlcToNc <-> Inputs/FromPlc
//   (this object) <-> NC-Task 1 SAF/Axes/Axis 4
//     PlcTask Inputs/MAIN.mover[1].fbSwivelMovement.stAxisZ.NcToPlc <-> Outputs/ToPlc
//     PlcTask Outputs/MAIN.mover[1].fbSwivelMovement.stAxisZ.PlcToNc <-> Inputs/FromPlc
//   (this object) <-> NC-Task 1 SAF/Axes/Axis 5
//     PlcTask Inputs/MAIN.mover[1].fbSwivelMovement.stAxisB.NcToPlc <-> Outputs/ToPlc
//     PlcTask Outputs/MAIN.mover[1].fbSwivelMovement.stAxisB.PlcToNc <-> Inputs/FromPlc
//   (this object) <-> NC-Task 1 SAF/Axes/Axis a
//     PlcTask Inputs/MAIN.mover[2].fbShakeMovement.stAxisA.NcToPlc <-> Outputs/ToPlc
//     PlcTask Outputs/MAIN.mover[2].fbShakeMovement.stAxisA.PlcToNc <-> Inputs/FromPlc
//   (this object) <-> NC-Task 1 SAF/Axes/Axis b
//     PlcTask Inputs/MAIN.mover[2].fbShakeMovement.stAxisB.NcToPlc <-> Outputs/ToPlc
//     PlcTask Outputs/MAIN.mover[2].fbShakeMovement.stAxisB.PlcToNc <-> Inputs/FromPlc
//   (this object) <-> NC-Task 1 SAF/Axes/Axis x
//     PlcTask Inputs/MAIN.mover[2].fbShakeMovement.stAxisX.NcToPlc <-> Outputs/ToPlc
//     PlcTask Outputs/MAIN.mover[2].fbShakeMovement.stAxisX.PlcToNc <-> Inputs/FromPlc
//   (this object) <-> NC-Task 1 SAF/Axes/Axis y
//     PlcTask Inputs/MAIN.mover[2].fbShakeMovement.stAxisY.NcToPlc <-> Outputs/ToPlc
//     PlcTask Outputs/MAIN.mover[2].fbShakeMovement.stAxisY.PlcToNc <-> Inputs/FromPlc
//   (this object) <-> NC-Task 1 SAF/Axes/MasterShake
//     PlcTask Inputs/MAIN.mover[2].fbShakeMovement.stAxisMaster.NcToPlc <-> Outputs/ToPlc
//     PlcTask Outputs/MAIN.mover[2].fbShakeMovement.stAxisMaster.PlcToNc <-> Inputs/FromPlc
//   (this object) <-> XPlanar MC Project/Axes/Mover4220_1
//     PlcTask Inputs/MAIN.mover[1].fbMoverStandard.stMoverRef.MCTOPLC/ACT <-> McToPlc/ACT
//     PlcTask Inputs/MAIN.mover[1].fbMoverStandard.stMoverRef.MCTOPLC/COORDMODE <-> McToPlc/COORDMODE
//     PlcTask Inputs/MAIN.mover[1].fbMoverStandard.stMoverRef.MCTOPLC/SET <-> McToPlc/SET
//     PlcTask Inputs/MAIN.mover[1].fbMoverStandard.stMoverRef.MCTOPLC/SETONTRACK <-> McToPlc/SETONTRACK
//     PlcTask Inputs/MAIN.mover[1].fbMoverStandard.stMoverRef.MCTOPLC/STD <-> McToPlc/STD
//     PlcTask Outputs/MAIN.mover[1].fbMoverStandard.stMoverRef.PLCTOMC/STD <-> PlcToMc/STD
//   (this object) <-> XPlanar MC Project/Axes/Mover4220_2
//     PlcTask Inputs/MAIN.mover[2].fbMoverStandard.stMoverRef.MCTOPLC/ACT <-> McToPlc/ACT
//     PlcTask Inputs/MAIN.mover[2].fbMoverStandard.stMoverRef.MCTOPLC/COORDMODE <-> McToPlc/COORDMODE
//     PlcTask Inputs/MAIN.mover[2].fbMoverStandard.stMoverRef.MCTOPLC/SET <-> McToPlc/SET
//     PlcTask Inputs/MAIN.mover[2].fbMoverStandard.stMoverRef.MCTOPLC/SETONTRACK <-> McToPlc/SETONTRACK
//     PlcTask Inputs/MAIN.mover[2].fbMoverStandard.stMoverRef.MCTOPLC/STD <-> McToPlc/STD
//     PlcTask Outputs/MAIN.mover[2].fbMoverStandard.stMoverRef.PLCTOMC/STD <-> PlcToMc/STD
//   (this object) <-> XPlanar MC Project/Groups/Group3 (Planar Track)
//     PlcTask Inputs/MAIN.Track8.stTrackRef.MCTOPLC_STD <-> McToPlc/STD

CONFIGURATION MoXX_2TilesDemo
    RESOURCE PLC ON TwinCAT3
        TASK PlcTask(INTERVAL := T#10ms, PRIORITY := 6);
        PROGRAM MAIN WITH PlcTask : MAIN;
    END_RESOURCE
END_CONFIGURATION

// ---- GVLs/GVL10_VAR_PRG.TcGVL
(* Variables for program blocks *)
VAR_GLOBAL PERSISTENT
	
	nPowerFailureCounter					:UINT;
	
END_VAR
VAR_GLOBAL
	
	(* PLC start detected *)
	bFirstCycleDetected						:BOOL;
	bMachineSequenzAktiv					:BOOL;		(* PLC startup done (LED test) program in cyclic mode *)

	(* Clock generator *)
	bClock500ms								:BOOL;		(* Clock 500ms on/off *)
	bClock1s								:BOOL;		(* Clock 1s on/off *)
	bClock2s								:BOOL;		(* Clock 2s on/off *)
	bRisingEdge500ms						:BOOL;		(* Rising edge all 500ms over one cycle *)
	bRisingEdge1s							:BOOL;		(* Edge after 1s over a cycle *)
	bRisingEdge2s							:BOOL;		(* Edge after 2s over a cycle *)

END_VAR
(* End *)

// ---- POUs/CustomerTemplates/GCode/I_GCode.TcIO
INTERFACE I_GCode

PROPERTY P_Return : REFERENCE to ST_CommandReturn
GET
END_GET
END_PROPERTY

METHOD StartMovement
VAR_INPUT
	sFilePath	: STRING;
END_VAR
END_METHOD

END_INTERFACE

// ---- POUs/CustomerTemplates/SwivelMovement/I_SwivelMovement.TcIO
INTERFACE I_SwivelMovement

PROPERTY P_Return : REFERENCE to ST_CommandReturn
GET
END_GET
END_PROPERTY

METHOD StartMovement
VAR_INPUT
	NumCycles		: UINT;
	Velo			: LREAL;
END_VAR
END_METHOD

END_INTERFACE

// ---- POUs/CustomerTemplates/Shake/I_ShakeMovement.TcIO
INTERFACE I_ShakeMovement

PROPERTY P_Return : REFERENCE to ST_CommandReturn
GET
END_GET
END_PROPERTY

METHOD StartMovement
VAR_INPUT
	NumCycles		: UINT;
	Velo			: LREAL;
END_VAR
END_METHOD

END_INTERFACE

// ---- POUs/I_MoverApplication.TcIO
INTERFACE I_MoverApplication

METHOD Cycle
END_METHOD

PROPERTY P_nMoverIndex : INT
GET
END_GET
SET
END_SET
END_PROPERTY

PROPERTY P_nTrackId : UDINT
GET
END_GET
SET
END_SET
END_PROPERTY

PROPERTY std : I_XPlanarMoverStandard
GET
END_GET
SET
END_SET
END_PROPERTY

END_INTERFACE

// ---- POUs/MAIN.TcPOU
PROGRAM MAIN
VAR
	// button
	IbSwitch		AT%I*	: BOOL;
	IbSwitchRestart	AT%I*	: BOOL;
	ObLamp			AT%Q*	: BOOL;	
	fbBlinker				: FB_Blinker;
	tcRestart 				: TC_Restart;

	nState 					: INT;
	mover					: ARRAY[1..2] OF FB_MoverApplication;
	ipMover					: ARRAY[1..2] OF I_MoverApplication;
	_ipMover				: ARRAY[1..2] OF I_MoverApplication;	
	cmdFb					: MC_PlanarFeedback;
	TargetPos				: PositionXYC;
	StartPos				: ARRAY[1..2] OF PositionXYC;
	Track8					: FB_TrackStandard;
	nStateTrackInit 		: INT;
	pstart					: REFERENCE TO PositionXYC;
	pend					: REFERENCE TO PositionXYC;
	pposition				: REFERENCE TO PositionXYC;
	start					: PositionXYC;
	end						: PositionXYC;
	position				: PositionXYC;
	
	
	
	// pattern Eight
	
	fSpeedEight 			: LREAL := 750;
	nCntEights				: INT;
	
	// Pattern Print
	nCnt					: INT;
	nStateP_Print			: INT;
	fYPos					: LREAL;
	
	// Pattern Rotation
	fCTargetPos				: LREAL;
	fRotCnt					: INT := 0;
	stMoveCOptions			: ST_MoveCOptions;
	stMoveCOptions2			: ST_MoveCOptions;
	nStateP_Rotation		: INT;
	
	// EIGHT
	StartPosEight			: ARRAY[1..2] OF PositionXYC;
	nStateP_Eight			: INT;
	
	// Pattern tilt
	nStateP_Tilt			: INT;
	
	
	// log
	fbWriteLog				: FB_WriteLog;
	tonTimer				: TON;
	nStateLog				: INT;
	stDiagData				: ST_CoeDriveDiagData;
	TilePower 				: UINT;
	nTemp1 					: UINT;
	nTemp2 					: UINT;
	nTemp3 					: UINT;
	nTemp4 					: UINT;
	nTemp5 					: UINT;
	//utility
	fbEnvironment			: FB_TcIoXPlanarEnvironment;
	ipXpu					: I_TcIoXPlanarProcessingUnit;
	fbXPlanarUtilityVisu	: FB_XPlanarUtilityVisu;
	nStateInitXpu			: INT;
	
	
	fPosX					: LREAL;
	fPosY					: LREAL;
	_Position				: PositionXYC;
	fTrackPos				: LREAL;
	fTrackLength			: LREAL;
	
	//shutdown
	fbDelay					:TON;	
	fbShutdown				:NT_SHUTDOWN;
	tDelay					:TIME := T#3000MS;
	bStartShutdown			:BOOL;
END_VAR

mover[1].Cycle();
mover[2].Cycle();
//ObLamp :=  IbSwitch;

fbBlinker(
	bStart 			:= (nstate > 10),
	tTurnOffDelay 	:= T#750MS,
	tTurnOnDelay	:= T#750MS,
	bLed			=> ObLamp);

actShutdown();

tcRestart(
	NETID:= , 
	RESTART:= IbSwitchRestart AND NOT bStartShutdown, 
	TMOUT:= , 
	BUSY=> , 
	ERR=> , 
	ERRID=> );

CASE nstate OF
	
-10:
	mover[1].std.Disable('');
	mover[2].std.Disable('');
	nstate := -9;	
	
-9:
	IF IbSwitch THEN
		nstate := 0;
	END_IF	

-2:
	mover[1].std.Reset('');
	mover[2].std.Reset('');
	nstate := -1;
-1:
	IF 	mover[1].std.P_Reset.Done
		AND mover[2].std.P_Reset.Done  THEN
		//nstate := 0;
	END_IF

0:
	IF IbSwitch THEN
		nstate := 1;
	END_IF
1:
	mover[1].std.Enable('');
	mover[2].std.Enable('');
	nstate := 2;
2:
	IF mover[1].std.P_Enable.Done
		AND mover[2].std.P_Enable.Done THEN
		nstate := 5;
	END_IF


5:
	IF mover[1].std.P_ActPosition.y < mover[2].std.P_ActPosition.y THEN
		ipMover[1] := mover[1];	
		ipMover[2] := mover[2];	
	ELSE
		ipMover[1] := mover[2];	
		ipMover[2] := mover[1];	
	END_IF
	nstate := 10;
	
10:
	StartPos[1].SetValuesXYC(120,120,0);
	StartPos[2].SetValuesXYC(120,360,0);
	nstate := 12;
	
	
12:

		nstate := 13;

13:
	Mover[1].std.MoveZ('',2.0,10,1000,1000,1000);
	Mover[2].std.MoveZ('',4.0,100,1000,1000,1000);
	nState := 14;
14:
	IF ipMover[1].std.P_MoveZ.Done 
		AND  ipMover[2].std.P_MoveZ.Done THEN
		nstate := 15;
	END_IF		
	
	
15:
	ipMover[1].std.MoveToPosition('',startpos[1],2000,20000,20000,2000000);
	ipMover[2].std.MoveToPosition('',startpos[2],2000,20000,20000,2000000);	

	nstate := 16;

16:
	   Mover[1].Swivel.StartMovement(5,250);
	   Mover[2].Shake.StartMovement(10,500);
	   nstate := 17;
	 
17:
		IF	  mover[1].Swivel.P_Return.Done 
			AND mover[2].Shake.P_Return.Done THEN
			
		
			Mover[2].std.MoveZ('',2.0,100,1000,1000,1000);
	 		nstate := 20;
	 END_IF


20:
	IF ipMover[1].std.P_MoveToPosition.Done 
		AND ipMover[2].std.P_MoveToPosition.Done THEN
		nStateP_Eight := 1;
		nstate := 21;
	END_IF		

21:
	IF 	nStateP_Eight = 0 THEN
		nstate := 30;
	END_IF
	
30:
	nStateP_Rotation := 1;
	nstate := 31;
31:
	IF 	nStateP_Rotation = 0 THEN
		nstate := 40;
	END_IF
	
	
40:

	nStateP_Tilt := 1;
	nstate := 41;
	
41:
	IF nStateP_Tilt = 0 THEN
		nstate := 100;
	END_IF

	





100:
IF IbSwitch THEN
	nstate := 15;
ELSE
	nstate :=  -10;
END_IF
	

	
END_CASE
	// Eight
	CASE 	nStateP_Eight OF
		
	1:
		StartPosEight[1].SetValuesXYC(60,60,0);
		StartPosEight[2].SetValuesXYC(180,180,0);
		nStateP_Eight := 2;
	2:
		ipMover[1].std.MoveToPosition('',StartPosEight[1],2000,20000,20000,2000000);
		ipMover[2].std.MoveToPosition('',StartPosEight[2],2000,20000,20000,2000000);	
	
		nStateP_Eight := 3;
	3:
		IF ipMover[1].std.P_MoveToPosition.Done 	
			AND ipMover[2].std.P_MoveToPosition.Done THEN
			nStateP_Eight := 10;
		END_IF		
		
		
	10:
		nCntEights := 0;
		ipMover[1].std.JoinTrack('',track8,1000,3000,10000,0);
		ipMover[2].std.JoinTrack('',track8,1000,3000,10000,0);
		nStateP_Eight := 12;
	
	12:
		IF ipMover[1].std.P_JoinTrack.Done 
			AND ipMover[2].std.P_JoinTrack.Done THEN
			nStateP_Eight := 13;
		END_IF
		
	13:
		 ipMover[1].std.MoveOnTrack('',track8,864 +(5*fTrackLength),fSpeedEight,5000,500000,30,Tc3_Mc3PlanarMotion.MC_DIRECTION.mcDirectionNonModulo);
		 ipMover[2].std.MoveOnTrack('',track8,651+(5*fTrackLength),fSpeedEight,5000,500000,30,Tc3_Mc3PlanarMotion.MC_DIRECTION.mcDirectionNonModulo);
		nStateP_Eight := 14;
		

		14:
		IF ipMover[1].std.P_MoveOnTrack.Done 	
			AND ipMover[2].std.P_MoveOnTrack.Done THEN
			nStateP_Eight := 20;
		END_IF		
		
		20:
		ipMover[1].std.LeaveTrack('',StartPosEight[1],1000,5000,5000,50000,0);
		ipMover[2].std.LeaveTrack('',StartPosEight[2],1000,5000,5000,50000,0);	
		nStateP_Eight := 21;
	
		21:
		IF ipMover[1].std.P_LeaveTrack.Done 
			AND ipMover[2].std.P_LeaveTrack.Done  THEN
			nStateP_Eight := 30;
		END_IF
		
		
		
		
	30:
		StartPosEight[1].SetValuesXYC(60,480-60,0);
		StartPosEight[2].SetValuesXYC(180,60,0);

		nStateP_Eight := 31;
	31:
		ipMover[1].std.MoveToPosition('',StartPosEight[1],2000,20000,20000,2000000);
		ipMover[2].std.MoveToPosition('',StartPosEight[2],2000,20000,20000,2000000);	
	
		nStateP_Eight := 32;
	32:
		IF ipMover[1].std.P_MoveToPosition.Done 	
			AND ipMover[2].std.P_MoveToPosition.Done THEN
			nStateP_Eight := 35;
		END_IF		
		

	35:	
		StartPosEight[1].SetValuesXYC(60,60,0);
		StartPosEight[2].SetValuesXYC(180,480-60,0);

		nStateP_Eight := 36;
	36:
		ipMover[1].std.MoveToPosition('',StartPosEight[1],2000,20000,20000,2000000);
		ipMover[2].std.MoveToPosition('',StartPosEight[2],2000,20000,20000,2000000);	
	
		nStateP_Eight := 37;
	37:
		IF ipMover[1].std.P_MoveToPosition.Done 	
			AND ipMover[2].std.P_MoveToPosition.Done THEN
			
			nCntEights := nCntEights +1;
			nStateP_Eight := 40;
		END_IF	
	40:
		IF nCntEights >= 5 THEN
			nStateP_Eight := 50;
		ELSE
			nStateP_Eight := 30;
		END_IF

	50:
		StartPosEight[1].SetValuesXYC(180,60,0);
		StartPosEight[2].SetValuesXYC(60,480-60,0);
		ipMover[1].std.MoveToPosition('',StartPosEight[1],2000,20000,20000,2000000);
		ipMover[2].std.MoveToPosition('',StartPosEight[2],2000,20000,20000,2000000);	
	
		nStateP_Eight := 51;
	51:
		IF ipMover[1].std.P_MoveToPosition.Done 	
			AND ipMover[2].std.P_MoveToPosition.Done THEN
					nStateP_Eight := 52;
		END_IF
			
			
	52:
		_ipMover[1] := ipMover[1];
		_ipMover[2] := ipMover[2];
		
		ipMover[1] := _ipMover[2];
		ipMover[2] := _ipMover[1];

		nStateP_Eight := 55;

	55:
		IF nCntEights >= 10 THEN
			nStateP_Eight := 60;
		ELSE
			nStateP_Eight := 30;
		END_IF

	60:
		_ipMover[1] := ipMover[1];
		_ipMover[2] := ipMover[2];
		
		ipMover[1] := _ipMover[2];
		ipMover[2] := _ipMover[1];

		nStateP_Eight := 90;

	90:
	
		ipMover[1].std.MoveToPosition('',startpos[1],2000,20000,20000,2000000);
		ipMover[2].std.MoveToPosition('',startpos[2],2000,20000,20000,2000000);	
	
		nStateP_Eight := 91;
	91:
		IF ipMover[1].std.P_MoveToPosition.Done 
			AND ipMover[2].std.P_MoveToPosition.Done THEN
			nStateP_Eight := 0;
		END_IF	
	END_CASE

	
	
	
	
	
	
	
	
	
	
	
	
	
	
	
	
	
	
	
	
	// ROTATION
	CASE 	nStateP_Rotation OF
		
	1:
	
		StartPos[1].SetValuesXYC(120,120,0);
		StartPos[2].SetValuesXYC(120,360,0);
		fCTargetPos := 10;
		ipmover[1].std.MoveToPosition('',startpos[1],2000,20000,20000,2000000);
		ipmover[2].std.MoveToPosition('',startpos[2],2000,20000,20000,2000000);
		nStateP_Rotation := 2;
	2:
		IF ipmover[1].std.P_MoveToPosition.Done
			AND ipmover[2].std.P_MoveToPosition.Done THEN
			nStateP_Rotation := 10;
		END_IF
	10:
		stMoveCOptions.additionalTurns := 0;
		stMoveCOptions.direction := Tc3_Mc3PlanarMotion.  MC_DIRECTION.mcDirectionNegative;
		ipmover[1].std.MoveC('',360-fCTargetPos,360*(fCTargetPos/5),500,500,1000,stMoveCOptions);
		stMoveCOptions2.additionalTurns := 0;
		stMoveCOptions2.direction := Tc3_Mc3PlanarMotion.MC_DIRECTION.mcDirectionPositive;
		ipmover[2].std.MoveC('',fCTargetPos,360*(fCTargetPos/5),500,500,1000,stMoveCOptions2);
		nStateP_Rotation := 11;
	11:
		IF ipmover[1].std.P_MoveC.Done 
			AND ipmover[2].std.P_MoveC.Done THEN
		
				nStateP_Rotation := 15;
			END_IF

	15:
		stMoveCOptions.additionalTurns := 0;
		stMoveCOptions.direction := Tc3_Mc3PlanarMotion.MC_DIRECTION.mcDirectionPositive;
		ipmover[1].std.MoveC('',fCTargetPos,360*(fCTargetPos/5),500,500,1000,stMoveCOptions);
		stMoveCOptions2.additionalTurns := 0;
		stMoveCOptions2.direction := Tc3_Mc3PlanarMotion.MC_DIRECTION.mcDirectionNegative;		
		ipmover[2].std.MoveC('',360-fCTargetPos,360*(fCTargetPos/5),500,500,1000,stMoveCOptions2);
		nStateP_Rotation := 16;
	16:
		IF ipmover[1].std.P_MoveC.Done THEN
				fCTargetPos := fCTargetPos + 30;
				nStateP_Rotation := 20;
		END_IF

		IF 	fCTargetPos >= 160 THEN
			nStateP_Rotation := 30;
		END_IF

	20:
		IF 	fCTargetPos > 180 THEN
			nStateP_Rotation := 30;
		ELSE
			nStateP_Rotation := 10;
		END_IF
		
		
	30:
		stMoveCOptions.additionalTurns := 30;
		stMoveCOptions2.additionalTurns := 30;
		stMoveCOptions.direction := Tc3_Mc3PlanarMotion.MC_DIRECTION.mcDirectionNegative;
		stMoveCOptions2.direction := Tc3_Mc3PlanarMotion.MC_DIRECTION.mcDirectionPositive;
		ipmover[1].std.MoveC('',0,8*360,1000,100000,100000,stMoveCOptions);
		ipmover[2].std.MoveC('',0,8*360,1000,100000,100000,stMoveCOptions2);
		nStateP_Rotation := 31;
		
	31:
			IF ipmover[1].std.P_MoveC.Done
				AND ipmover[1].std.P_MoveC.Done THEN
				
				nStateP_Rotation := 0;
			END_IF	
			
		
	END_CASE

(*
	// PRINTER
	CASE nStateP_Print OF	
		
	0:
	
	1:
		nStateP_Print := 10;
		fYPos := 0;
	10:
		TargetPos.SetValuesXYC(60,60+fYPos,0);
		mover[1].std.MoveToPosition('',targetpos,2000,20000,20000,2000000);
		nStateP_Print := 11;
	
		
	11:	
		IF mover[1].std.P_MoveToPosition.Done THEN
			nStateP_Print := 12;
		END_IF
		
	12:
		TargetPos.SetValuesXYC(420,60+fYPos,0);
		mover[1].std.MoveToPosition('',targetpos,2000,20000,20000,2000000);
		nStateP_Print := 13;
	
		
	13:	
		IF mover[1].std.P_MoveToPosition.Done THEN
			fYPos := fYPos+1;
			nStateP_Print := 14;
		END_IF	
		
	14:
		TargetPos.SetValuesXYC(420,60+fYPos,0);
		mover[1].std.MoveToPosition('',targetpos,2000,20000,20000,2000000);
		nStateP_Print := 15;
	15:
		IF mover[1].std.P_MoveToPosition.Done THEN
			fYPos := fYPos+5;
			nStateP_Print := 16;
		END_IF		
	16:
		IF fYPos > 120 THEN
			nStateP_Print := 20;
		ELSE
			nStateP_Print := 10;
		END_IF
	20:
		mover[1].std.MoveToPosition('',startpos[1],2000,20000,20000,2000000);
		nStateP_Print := 21;
	21:
		IF mover[1].std.P_MoveToPosition.Done THEN
			nStateP_Print := 0;
		END_IF
	
	END_CASE	

*)
	
	
	
CASE nStateP_Tilt	OF
	


1:
	ipMover[1].std.MoveZ('',5.0,1000,2000,2000,20000);
	ipMover[2].std.MoveZ('',5.0,1000,2000,2000,20000);
	nStateP_Tilt := 2;

2:	
	IF ipMover[1].std.P_MoveZ.Done 
			AND ipMover[2].std.P_MoveZ.Done THEN
			nStateP_Tilt := 5;
	END_IF	
	
	
5:
	ipMover[1].std.Movea('',2.5,1000,2000,2000,20000);
	ipMover[2].std.Movea('',-2.5,1000,2000,2000,20000);
	nStateP_Tilt := 6;

6: 
	IF ipMover[1].std.P_Movea.Done 
			AND ipMover[2].std.P_Movea.Done THEN
			nStateP_Tilt := 10;
	END_IF		
10:
	ipMover[1].std.Movea('',-2,1000,2000,2000,20000);
	ipMover[2].std.Movea('',2,1000,2000,2000,20000);
	
	ipMover[1].std.Moveb('',2,1000,2000,2000,20000);
	ipMover[2].std.Moveb('',-2,1000,2000,2000,20000);
	nStateP_Tilt := 11;

11:
	IF ipMover[1].std.P_Movea.Done 
			AND ipMover[2].std.P_Movea.Done THEN
			nStateP_Tilt := 15;
	END_IF	
15:
	//ipMover[1].std.Movea('',3,1000,2000,2000,20000);
	//ipMover[2].std.Movea('',-3,1000,2000,2000,20000);
	
	ipMover[1].std.Moveb('',-2,1000,2000,2000,20000);
	ipMover[2].std.Moveb('',2,1000,2000,2000,20000);
	
	nStateP_Tilt := 20;	
20:	
	IF ipMover[1].std.P_Moveb.Done 
			AND ipMover[2].std.P_Moveb.Done THEN
			nStateP_Tilt := 25;
	END_IF	

25:	
	ipMover[1].std.Movea('',0,1000,2000,2000,20000);
	ipMover[2].std.Movea('',0,1000,2000,2000,20000);
	nStateP_Tilt := 26;
26:
	IF ipMover[1].std.P_Movea.Done 
			AND ipMover[2].std.P_Movea.Done THEN
			nStateP_Tilt := 27;
	END_IF

27:
	ipMover[1].std.Moveb('',0,1000,2000,2000,20000);
	ipMover[2].std.Moveb('',0,1000,2000,2000,20000);	

	nStateP_Tilt := 28;
	
28:
	IF ipMover[1].std.P_Moveb.Done 
			AND ipMover[2].std.P_Moveb.Done THEN
			nStateP_Tilt := 30;
	END_IF

	
30:			
	ipMover[1].std.MoveZ('',2.0,1000,2000,2000,20000);
	ipMover[2].std.MoveZ('',2.0,1000,2000,2000,20000);		
			nStateP_Tilt := nStateP_Tilt +1;

31:
	IF ipMover[1].std.P_MoveZ.Done 
			AND ipMover[2].std.P_MoveZ.Done THEN
			nStateP_Tilt := 0;
	END_IF	
	
END_CASE
	
	
	
	
	
	
	
	
	
	
	
	
	

CASE nStateInitXpu OF
0: // init environment
		IF fbEnvironment.Init(TRUE) THEN
			fbEnvironment.Init(FALSE);
			nStateInitXpu:=1;
		END_IF

1: // init Visu
	fbXPlanarUtilityVisu.Environment := fbEnvironment;
	nStateInitXpu := 3;	

3:
	ipXpu := fbEnvironment.XpuTcIo(1);
	nStateInitXpu := 4;
	
ELSE // call Visu
	fbXPlanarUtilityVisu.Cycle();
END_CASE

IF nStateInitXpu <> 4 THEN
RETURN;
END_IF

(*
fbWriteLog(sPath:='c:\templog\log.txt' , bErrorAcknowledge:= );


tonTimer(IN:= , PT:=T#60S , Q=> , ET=> );

CASE nstatelog OF
	
0:
tonTimer(IN:=TRUE);
	IF tonTimer.Q THEN
		nstatelog := 1;
	END_IF

1:
IF ipXpu.TileCoE(1,1).DiagData.Update() THEN
	TilePower := LREAL_TO_UINT(ipXpu.TileTcIo(1,1).GetObservedTilePower());
	stDiagData.TemperatureCenter := ipXpu.TileCoE(1,1).DiagData.TemperatureCenter;
	stDiagData.TemperatureNorth := ipXpu.TileCoE(1,1).DiagData.TemperatureNorth;
	stDiagData.TemperatureEast := ipXpu.TileCoE(1,1).DiagData.TemperatureEast;
	stDiagData.TemperatureSouth := ipXpu.TileCoE(1,1).DiagData.TemperatureSouth;
	stDiagData.TemperatureWest := ipXpu.TileCoE(1,1).DiagData.TemperatureWest;
	nstatelog := 0;
	tonTimer(IN:=FALSE);
	fbWriteLog.M_AddLogg(CONCAT(UINT_TO_STRING(stDiagData.TemperatureCenter),CONCAT(';',CONCAT(UINT_TO_STRING(stDiagData.TemperatureNorth),CONCAT(';',CONCAT(UINT_TO_STRING(stDiagData.TemperatureEast),CONCAT(';',CONCAT(UINT_TO_STRING(stDiagData.TemperatureSouth),CONCAT(';',CONCAT(UINT_TO_STRING(stDiagData.TemperatureWest),CONCAT(';',UINT_TO_STRING(TilePower))))))))))));


END_IF

END_CASE

*)






CASE nStateTrackInit OF
	
0:
	track8.Reset();
	
	pstart REF= start;
	pend REF= end;
	pposition REF= position;
	
	nStateTrackInit := 1;
1:
	IF track8.P_Reset.done THEN
		nStateTrackInit := 2;
	END_IF
2:
	start.SetValuesXYC(120-20,240-1,0);
	end.SetValuesXYC(120+20,240+1,0);
	track8.AppendLine(start,end);

	pposition.SetValuesXYC(180,300,0);
//	track8.AppendPoint(pposition);
	
	// rechts oben
	start.SetValuesXYC(240-60,360-1,0);
	end.SetValuesXYC(240-60,360+20,0);	
	track8.AppendLine(start,end);
	
	pposition.SetValuesXYC(420,420,0);
//	track8.AppendPoint(pposition);

	// rechts mitte
	start.SetValuesXYC(120+1,480-60,0);
	end.SetValuesXYC(120-1,480-60,0);	
	track8.AppendLine(start,end);
	
	pposition.SetValuesXYC(60,420,0);
//	track8.AppendPoint(pposition);
	
	// rechts unten
	start.SetValuesXYC(60,360+20,0);
	end.SetValuesXYC(60,360-1,0);	
	track8.AppendLine(start,end);	
	
	pposition.SetValuesXYC(60,300,0);
//	track8.AppendPoint(pposition);

	// kreuz von rechts unten nach links oben
	start.SetValuesXYC(120-20,240+1,0);
	end.SetValuesXYC(120+20,240-1,0);
	track8.AppendLine(start,end);	
	
//	pposition.SetValuesXYC(180,180,0);
//	track8.AppendPoint(pposition);
	
	// links oben
	start.SetValuesXYC(240-60,120+1,0);
	end.SetValuesXYC(240-60,120-20,0);	
	track8.AppendLine(start,end);

	pposition.SetValuesXYC(180,60,0);
//	track8.AppendPoint(pposition);
	
	// libks mitte
	start.SetValuesXYC(120+1,60,0);
	end.SetValuesXYC(120-1,60,0);	
	track8.AppendLine(start,end);
	
	pposition.SetValuesXYC(60,60,0);
//	track8.AppendPoint(pposition);
	
	//links unten
	start.SetValuesXYC(60,120-20,0);
	end.SetValuesXYC(60,120+1,0);	
	track8.AppendLine(start,end);
	
	pposition.SetValuesXYC(60,180,0);
//	track8.AppendPoint(pposition);

	track8.CloseLoop();
	nStateTrackInit := 3;
3:
	IF track8.P_CloseLoop.Done THEN
		nStateTrackInit := 4;
	END_IF
4:
	Track8.Enable();
	nStateTrackInit := 5;
5:
	IF Track8.P_Enable.Done THEN
		nStateTrackInit := 6;
	END_IF
END_CASE
track8.Cycle();




fTrackLength := track8.GetLength();

track8.GetMoverPositionAt(fTrackPos,_Position);
fPosX := _Position.x;
fPosY := _Position.y;

fTrackPos := fTrackPos +1;
IF fTrackPos >= fTrackLength THEN
	fTrackPos := 1;
END_IF

ACTION actShutdown:
//act Shutdown

	IF TwinCAT_SystemInfoVarList._TaskInfo[GETCURTASKINDEXEX()].FirstCycle
		AND IbSwitchRestart
	THEN
		bStartShutdown	:= TRUE;
	END_IF

	fbDelay(
		IN := IbSwitchRestart,
		PT := tDelay);
		
	fbShutdown(
		START := fbDelay.Q);	



//End
END_ACTION

METHOD Shutdown : BOOL
VAR_INPUT
	bExecute		:BOOL;
END_VAR
VAR_INST


END_VAR
// mShutdown




//End
END_METHOD

END_PROGRAM

// ---- POUs/10_GeneralPlcBlocks/Components/FB_Blinker.TcPOU
FUNCTION_BLOCK FB_Blinker
VAR_INPUT

	bStart									:BOOL;
	tTurnOnDelay							:TIME;
	tTurnOffDelay							:TIME;

END_VAR
VAR_OUTPUT

	bLed									:BOOL;

END_VAR
VAR

	fbTimer1								:TON;
	fbTimer2								:TON;

END_VAR
(* End *)

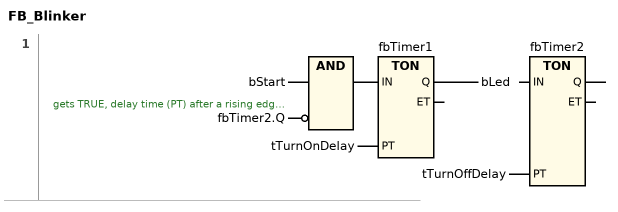
// NETWORK 1
//   fbTimer2.Q: gets TRUE, delay time (PT) after a rising edge at IN
fbTimer1(IN := bStart AND NOT fbTimer2.Q, PT := tTurnOnDelay); // TON
bLed := fbTimer1.Q;
fbTimer2(IN := fbTimer1.Q, PT := tTurnOffDelay); // TON

END_FUNCTION_BLOCK

// ---- POUs/FB_MoverApplication.TcPOU
FUNCTION_BLOCK FB_MoverApplication IMPLEMENTS I_MoverApplication
VAR
	ipMoverStandard	: I_XPlanarMoverStandard;
	fbMoverStandard	: FB_XPlanarMoverStandard;

	
	nMoverIndex		: INT;
	
	nTrackId		: UDINT;
	
	// customer Data
	bIsLoaded		: BOOL;	
		
		
	// customer templates
	fbSwivelMovement 	: FB_SwivelMovement;
	ipSwivelMovement	: I_SwivelMovement;	
	
	fbShakeMovement 	: FB_ShakeMovement;
	ipShakeMovement		: I_ShakeMovement;		
	
	fbGCode			: FB_GCode;
	ipGCode			: I_GCode;
	
	
		
END_VAR

VAR_OUTPUT
	VisuPos	: MoverVector;
END_VAR

METHOD Cycle
ipMoverStandard := fbMoverStandard;


IF std <> 0 THEN
	std.cycle();
	VisuPos := std.P_ActPosition;
END_IF



// additional functionality
ipSwivelMovement := fbSwivelMovement;
fbSwivelMovement(ipMover := ipMoverStandard);
fbSwivelMovement.Cycle();


ipShakeMovement := fbShakeMovement;
fbShakeMovement(ipMover := ipMoverStandard);
fbShakeMovement.Cycle();

ipGCode := fbGCode;
fbGCode(ipMover := ipMoverStandard);
fbGCode.Cycle();
END_METHOD

PROPERTY GCode : I_GCode
GET
IF ipGCode <> 0 THEN
	GCode := ipGCode;	
END_IF
END_GET
SET
ipGCode := GCode;
END_SET
END_PROPERTY

PROPERTY P_nMoverIndex : INT
GET
P_nMoverIndex := nMoverIndex;
END_GET
SET
nMoverIndex := P_nMoverIndex;
END_SET
END_PROPERTY

PROPERTY P_nTrackId : UDINT
GET
P_nTrackId := nTrackId;
END_GET
SET
nTrackId := P_nTrackId;
END_SET
END_PROPERTY

PROPERTY Shake : I_ShakeMovement
GET
IF ipShakeMovement <> 0 THEN
	Shake := ipShakeMovement;	
END_IF
END_GET
SET
ipShakeMovement := Shake;
END_SET
END_PROPERTY

PROPERTY std : I_XPlanarMoverStandard
GET
IF ipMoverStandard <> 0 THEN
	std := ipMoverStandard;	
END_IF
END_GET
SET
ipMoverStandard := std;
END_SET
END_PROPERTY

PROPERTY Swivel : I_SwivelMovement
GET
IF ipSwivelMovement <> 0 THEN
	Swivel := ipSwivelMovement;	
END_IF
END_GET
SET
ipSwivelMovement := Swivel;
END_SET
END_PROPERTY

END_FUNCTION_BLOCK

// ---- POUs/CustomerTemplates/SwivelMovement/FB_SwivelMovement.TcPOU
FUNCTION_BLOCK FB_SwivelMovement IMPLEMENTS I_SwivelMovement

VAR_INPUT

END_VAR

VAR

// NC 
	stAxisMaster	: AXIS_REF;
	stAxisZ			: AXIS_REF;
	stAxisB			: AXIS_REF;	
	stAxisX			: AXIS_REF;
	stAxisY			: AXIS_REF;

	mcPower			: MC_Power;
	
	mcMoveAbsZ		: MC_MoveAbsolute;
	mcMoveAbsX		: MC_MoveAbsolute;
	mcMoveAbsMaster	: MC_MoveAbsolute;
	
	mcSetPos		: MC_SetPosition;
	
	
	McCamIn			: MC_Camin;	
	McCamOut		: MC_CamOut;
	
	nState			: INT := -20;
	
	bStartCam		: BOOL;
	
	ExtSetPos		: MoverVector;
	ExtSetVelo		: MoverVector;
	ExtSetAcc		: MoverVector;
	

// parameters
	fAmpZ			: LREAL := 0;
	fAmpA			: LREAL := 2;	
	nNumCycles		: UINT := 1;
	nVeloMaster		: LREAL;
	
// internal
	bExecute		: BOOL;
	rtrigExecute 	: R_TRIG;
	stReturn		: ST_CommandReturn;
END_VAR



VAR_IN_OUT
	ipMover			: I_XPlanarMoverStandard;
END_VAR

{attribute 'hide'}
METHOD PROTECTED ccl_StartMovement
VAR_INPUT
END_VAR
CASE nState OF

-20:

McCamOut(
	Slave:= stAxisX, 
	Execute:= TRUE);
IF McCamOut.Done THEN
	McCamOut(
		Slave:= stAxisX, 
		Execute:= FALSE);	
	nState := nState+1;
END_IF
-19:
McCamOut(
	Slave:= stAxisY, 
	Execute:= TRUE);
IF McCamOut.Done THEN
	McCamOut(
		Slave:= stAxisY, 
		Execute:= FALSE);	
	nState := nState+1;
END_IF

-18:
McCamOut(
	Slave:= stAxisZ, 
	Execute:= TRUE);
IF McCamOut.Done THEN
	McCamOut(
		Slave:= stAxisZ, 
		Execute:= FALSE);	
	nState := nState+1;
END_IF
-17:
McCamOut(
	Slave:= stAxisB, 
	Execute:= TRUE);
IF McCamOut.Done THEN
	McCamOut(
		Slave:= stAxisB, 
		Execute:= FALSE);	
	nState := -15;
END_IF

-15:
		nState := -10;

-10:

	mcPower(
		Axis:= stAxisZ, 
		Enable:= TRUE , 
		Enable_Positive:= TRUE , 
		Enable_Negative:= TRUE );
	IF NOT stAxisZ.Status.Disabled THEN
		nState := -9;
	END_IF

-9:
	mcPower(
		Axis:= stAxisMaster, 
		Enable:= TRUE , 
		Enable_Positive:= TRUE , 
		Enable_Negative:= TRUE );
	IF NOT stAxisMaster.Status.Disabled THEN
		nState := -8;
	END_IF


-8:

		nState := -7;
	

-7:

		nState := -6;


-6:

		nState := 0;
	


0:

		nState := 10;

	
10:

	ipMover.EnableExternalSetpointGeneration('start ext. setpoint gen',MC_EXTERNAL_SET_POSITION_MODE.Relative);
nState := 11;

11:
	IF ipMover.P_EnableExternalSetpointGeneration.Done THEN
		nState := 30;
	END_IF
	


	
	
30:
	mcMoveAbsZ(
		Axis:= stAxisZ, 
		Execute:= TRUE, 
		Position:= -fAmpZ , 
		Velocity:= 50, 
		Acceleration:= 500, 
		Deceleration:= 500, 
		Jerk:= 1000 );	

	
	IF mcMoveAbsZ.Done THEN

		mcMoveAbsZ(
			Axis:= stAxisZ, 
			Execute:= FALSE);

		nState := 40;				
	END_IF
		


40:
	McCamIn(
		Master:=  stAxisMaster, 
		Slave:= stAxisZ , 
		Execute:= TRUE , 
		MasterOffset:= , 
		SlaveOffset:= , 
		MasterScaling:= , 
		SlaveScaling:= , 
		StartMode:= , 
		CamTableID:=1 , 
		BufferMode:= , 
		Options:= , 
		InSync=> , 
		Busy=> , 
		Active=> , 
		CommandAborted=> , 
		Error=> , 
		ErrorID=> );
	IF McCamIn.InSync THEN
		McCamIn(
			Master:=  stAxisMaster, 
			Slave:= stAxisZ , 
			Execute:= FALSE);
		nState := 50;
	END_IF

	
50:	
	mcMoveAbsMaster(
		Axis:= stAxisMaster, 
		Execute:= TRUE, 
		Position:=  nNumCycles*360.0, 
		Velocity:= nVeloMaster, 
		Acceleration:= 1000, 
		Deceleration:= 1000, 
		Jerk:= 1000 );
	IF mcMoveAbsMaster.Done THEN
			mcMoveAbsMaster(
				Axis:= stAxisMaster, 
				Execute:= FALSE);
			nState := nState +1;
	END_IF
	
51:
	McCamOut(
		Slave:= stAxisZ, 
		Execute:= TRUE);
	IF McCamOut.Done THEN
		McCamOut(
			Slave:= stAxisZ, 
			Execute:= FALSE);
		nState := nState +1;
	END_IF
	
52:

		nState := nState +1;

53:	

		nState := nState +1;

54:

		nState := nState +1;
	
	
55:
	mcMoveAbsZ(
		Axis:= stAxisZ, 
		Execute:= TRUE, 
		Position:= 0, 
		Velocity:= 50, 
		Acceleration:= 500, 
		Deceleration:= 500, 
		Jerk:= 1000 );	


	IF mcMoveAbsZ.Done THEN

		mcMoveAbsZ(
			Axis:= stAxisZ, 
			Execute:= FALSE);

		nState := 58;				
	END_IF


58:
	ipMover.DisableExternalSetpointGeneration('disable ext. setpoints');
	nState := nState +1;
59:
	IF ipMover.P_DisableExternalSetpointGeneration.Done THEN
		nState := nState +1;
	END_IF
	
60:
	mcSetPos(
	Axis:= stAxisMaster , 
	Execute:= TRUE,
	Position := 0);
	IF mcSetPos.Done THEN
		mcSetPos(
			Axis:= stAxisMaster , 
			Execute:= FALSE);
		nstate := 70;
	END_IF
	
70:
	bExecute := FALSE;
	stReturn.Active := FALSE;
	streturn.Done := TRUE;
	nstate := 0;


	
	
END_CASE


CASE nstate OF
	20..60:
		
	
		ExtSetPos.x := stAxisX.NcToPlc.SetPos; 
		ExtSetPos.y := stAxisY.NcToPlc.SetPos; 
		ExtSetPos.z := stAxisZ.NcToPlc.SetPos; 
		ExtSetPos.b := stAxisB.NcToPlc.SetPos;	
	
		ExtSetVelo.x := stAxisX.NcToPlc.SetVelo; 
		ExtSetVelo.y := stAxisY.NcToPlc.SetVelo; 
		ExtSetVelo.z := stAxisZ.NcToPlc.SetVelo; 
		ExtSetVelo.b := stAxisB.NcToPlc.SetVelo; 
	
		ExtSetAcc.x := stAxisX.NcToPlc.SetAcc; 
		ExtSetAcc.y := stAxisY.NcToPlc.SetAcc; 
		ExtSetAcc.z := stAxisZ.NcToPlc.SetAcc; 
		ExtSetAcc.b := stAxisB.NcToPlc.SetAcc; 		
		
	
		ipMover.SetExternalSetpointValues(ExtSetPos,ExtSetVelo,ExtSetAcc);
END_CASE


IF mcMoveAbsMaster.Error THEN
	mcMoveAbsMaster(Axis := stAxisMaster,Execute := FALSE);
	nstate := -50;
END_IF

IF mcMoveAbsMaster.Error 
	OR mcMoveAbsZ.error
	OR mcMoveAbsX.error
	OR mcPower.error
	OR mcSetPos.error
	OR McCamIn.error
	OR McCamOut.error THEN
	stReturn.Error := TRUE;
END_IF
END_METHOD

METHOD Cycle
VAR_INPUT
END_VAR
stAxisMaster.ReadStatus();
stAxisZ.ReadStatus();
stAxisB.ReadStatus();
stAxisX.ReadStatus();
stAxisY.ReadStatus();

rtrigExecute(CLK:= bExecute, Q=> );
IF rtrigExecute.Q THEN
	MEMSET(destAddr:=ADR(stReturn) , fillByte:=0 , n:=SIZEOF(stReturn) );
END_IF


IF bExecute THEN
	ccl_StartMovement();
END_IF
END_METHOD

PROPERTY P_Return : REFERENCE to ST_CommandReturn
GET
P_Return ReF= stReturn;
END_GET
END_PROPERTY

METHOD StartMovement
VAR_INPUT
	NumCycles		: UINT;
	Velo			: LREAL;
END_VAR
nNumCycles := numCycles;
nVeloMaster := Velo;

bExecute := TRUE;
END_METHOD

END_FUNCTION_BLOCK

// ---- POUs/CustomerTemplates/Shake/FB_ShakeMovement.TcPOU
FUNCTION_BLOCK FB_ShakeMovement IMPLEMENTS I_ShakeMovement

VAR_INPUT

END_VAR

VAR

// NC 
	stAxisMaster	: AXIS_REF;
	stAxisA			: AXIS_REF;
	stAxisB			: AXIS_REF;	
	stAxisX			: AXIS_REF;
	stAxisY			: AXIS_REF;

	mcPower			: MC_Power;
	
	mcMoveAbsA		: MC_MoveAbsolute;
	mcMoveAbsX		: MC_MoveAbsolute;
	mcMoveAbsMaster	: MC_MoveAbsolute;
	
	mcSetPos		: MC_SetPosition;
	
	
	McCamIn			: MC_Camin;	
	McCamOut		: MC_CamOut;
	
	nState			: INT := -20;
	
	bStartCam		: BOOL;
	
	ExtSetPos		: MoverVector;
	ExtSetVelo		: MoverVector;
	ExtSetAcc		: MoverVector;
	

// parameters
	fAmpX			: LREAL := 0;
	fAmpA			: LREAL := 0;	
	nNumCycles		: UINT := 1;
	nVeloMaster		: LREAL;
	
// internal
	bExecute		: BOOL;
	rtrigExecute 	: R_TRIG;
	stReturn		: ST_CommandReturn;
END_VAR



VAR_IN_OUT
	ipMover			: I_XPlanarMoverStandard;
END_VAR

{attribute 'hide'}
METHOD PROTECTED ccl_StartMovement
VAR_INPUT
END_VAR
CASE nState OF

-20:

McCamOut(
	Slave:= stAxisX, 
	Execute:= TRUE);
IF McCamOut.Done THEN
	McCamOut(
		Slave:= stAxisX, 
		Execute:= FALSE);	
	nState := nState+1;
END_IF
-19:
McCamOut(
	Slave:= stAxisY, 
	Execute:= TRUE);
IF McCamOut.Done THEN
	McCamOut(
		Slave:= stAxisY, 
		Execute:= FALSE);	
	nState := nState+1;
END_IF

-18:
McCamOut(
	Slave:= stAxisA, 
	Execute:= TRUE);
IF McCamOut.Done THEN
	McCamOut(
		Slave:= stAxisA, 
		Execute:= FALSE);	
	nState := nState+1;
END_IF
-17:
McCamOut(
	Slave:= stAxisB, 
	Execute:= TRUE);
IF McCamOut.Done THEN
	McCamOut(
		Slave:= stAxisB, 
		Execute:= FALSE);	
	nState := -15;
END_IF

-15:
		nState := -10;

-10:

	mcPower(
		Axis:= stAxisA, 
		Enable:= TRUE , 
		Enable_Positive:= TRUE , 
		Enable_Negative:= TRUE );
	IF NOT stAxisA.Status.Disabled THEN
		nState := -9;
	END_IF

-9:
	mcPower(
		Axis:= stAxisB, 
		Enable:= TRUE , 
		Enable_Positive:= TRUE , 
		Enable_Negative:= TRUE );
	IF NOT stAxisA.Status.Disabled THEN
		nState := -8;
	END_IF

-8:
	mcPower(
		Axis:= stAxisMaster, 
		Enable:= TRUE , 
		Enable_Positive:= TRUE , 
		Enable_Negative:= TRUE );
	IF NOT stAxisA.Status.Disabled THEN
		nState := -7;
	END_IF

-7:
	mcPower(
		Axis:= stAxisX, 
		Enable:= TRUE , 
		Enable_Positive:= TRUE , 
		Enable_Negative:= TRUE );
	IF NOT stAxisX.Status.Disabled THEN
		nState := -6;
	END_IF

-6:

	mcPower(
		Axis:= stAxisY, 
		Enable:= TRUE , 
		Enable_Positive:= TRUE , 
		Enable_Negative:= TRUE );
	IF NOT stAxisY.Status.Disabled THEN
		nState := 0;
	END_IF


0:

		nState := 10;

	
10:

	ipMover.EnableExternalSetpointGeneration('start ext. setpoint gen',MC_EXTERNAL_SET_POSITION_MODE.Relative);
	nState := nState+1;
	
11: 
	IF ipMover.P_EnableExternalSetpointGeneration.Done THEN
		nState := 30;
	END_IF
	


	
	
30:
	mcMoveAbsA(
		Axis:= stAxisA, 
		Execute:= TRUE, 
		Position:= -fAmpA , 
		Velocity:= 50, 
		Acceleration:= 500, 
		Deceleration:= 500, 
		Jerk:= 1000 );	

	
	mcMoveAbsX(
		Axis:= stAxisX, 
		Execute:= TRUE, 
		Position:= -fAmpX , 
		Velocity:= 50, 
		Acceleration:= 500, 
		Deceleration:= 500, 
		Jerk:= 1000 );	
	
	IF mcMoveAbsA.Done
		AND mcMoveAbsX.Done THEN

		mcMoveAbsA(
			Axis:= stAxisA, 
			Execute:= FALSE);
		mcMoveAbsX(
			Axis:= stAxisB, 
			Execute:= FALSE);
		nState := 40;				
	END_IF
		


40:
	McCamIn(
		Master:=  stAxisMaster, 
		Slave:= stAxisX , 
		Execute:= TRUE , 
		MasterOffset:= , 
		SlaveOffset:= , 
		MasterScaling:= , 
		SlaveScaling:= , 
		StartMode:= , 
		CamTableID:=4 , 
		BufferMode:= , 
		Options:= , 
		InSync=> , 
		Busy=> , 
		Active=> , 
		CommandAborted=> , 
		Error=> , 
		ErrorID=> );
	IF McCamIn.InSync THEN
		McCamIn(
			Master:=  stAxisMaster, 
			Slave:= stAxisX , 
			Execute:= FALSE);
		nState := nState +1;
	END_IF

41:
	McCamIn(
		Master:=  stAxisMaster, 
		Slave:= stAxisY , 
		Execute:= TRUE , 
		MasterOffset:= , 
		SlaveOffset:= , 
		MasterScaling:= , 
		SlaveScaling:= , 
		StartMode:= , 
		CamTableID:= 5, 
		BufferMode:= , 
		Options:= , 
		InSync=> , 
		Busy=> , 
		Active=> , 
		CommandAborted=> , 
		Error=> , 
		ErrorID=> );
	IF McCamIn.InSync THEN
		McCamIn(
			Master:=  stAxisMaster, 
			Slave:= stAxisY , 
			Execute:= FALSE);
		nState := nState +1;
	END_IF



42:
	McCamIn(
		Master:=  stAxisMaster, 
		Slave:= stAxisA , 
		Execute:= TRUE , 
		MasterOffset:= , 
		SlaveOffset:= , 
		MasterScaling:= , 
		SlaveScaling:= , 
		StartMode:= , 
		CamTableID:= 2, 
		BufferMode:= , 
		Options:= , 
		InSync=> , 
		Busy=> , 
		Active=> , 
		CommandAborted=> , 
		Error=> , 
		ErrorID=> );
	IF McCamIn.InSync THEN
		McCamIn(
			Master:=  stAxisMaster, 
			Slave:=  stAxisA, 
			Execute:= FALSE);
		nState := nState +1;
	END_IF

43:
	McCamIn(
		Master:=  stAxisMaster, 
		Slave:= stAxisB , 
		Execute:= TRUE , 
		MasterOffset:= , 
		SlaveOffset:= , 
		MasterScaling:= , 
		SlaveScaling:= , 
		StartMode:= , 
		CamTableID:= 3, 
		BufferMode:= , 
		Options:= , 
		InSync=> , 
		Busy=> , 
		Active=> , 
		CommandAborted=> , 
		Error=> , 
		ErrorID=> );
	IF McCamIn.InSync THEN
		McCamIn(
			Master:=  stAxisMaster, 
			Slave:=  stAxisB, 
			Execute:= FALSE);
		nState := 50;
	END_IF


50:

	mcMoveAbsMaster(
		Axis:= stAxisMaster, 
		Execute:= TRUE, 
		Position:=  nNumCycles*360.0, 
		Velocity:= nVeloMaster, 
		Acceleration:= 1000, 
		Deceleration:= 1000, 
		Jerk:= 1000 );
	IF mcMoveAbsMaster.Done THEN
			mcMoveAbsMaster(
				Axis:= stAxisMaster, 
				Execute:= FALSE);
			nState := nState +1;
	END_IF
	
51:
	McCamOut(
		Slave:= stAxisA, 
		Execute:= TRUE);
	IF McCamOut.Done THEN
		McCamOut(
			Slave:= stAxisA, 
			Execute:= FALSE);
		nState := nState +1;
	END_IF
	
52:

	McCamOut(
		Slave:= stAxisB, 
		Execute:= TRUE);
	IF McCamOut.Done THEN
		McCamOut(
			Slave:= stAxisB, 
			Execute:= FALSE);
		nState := nState +1;
	END_IF
53:	
	McCamOut(
		Slave:= stAxisX, 
		Execute:= TRUE);
	IF McCamOut.Done THEN
		McCamOut(
			Slave:= stAxisX, 
			Execute:= FALSE);
		nState := nState +1;
	END_IF
54:
	McCamOut(
		Slave:= stAxisY, 
		Execute:= TRUE);
	IF McCamOut.Done THEN
		McCamOut(
			Slave:= stAxisY, 
			Execute:= FALSE);
		nState := nState +1;
	END_IF	
	
55:
	mcMoveAbsA(
		Axis:= stAxisA, 
		Execute:= TRUE, 
		Position:= 0, 
		Velocity:= 50, 
		Acceleration:= 500, 
		Deceleration:= 500, 
		Jerk:= 1000 );	

	
	mcMoveAbsX(
		Axis:= stAxisX, 
		Execute:= TRUE, 
		Position:= 0 , 
		Velocity:= 50, 
		Acceleration:= 500, 
		Deceleration:= 500, 
		Jerk:= 1000 );	
	
	IF mcMoveAbsA.Done
		AND mcMoveAbsX.Done THEN

		mcMoveAbsA(
			Axis:= stAxisA, 
			Execute:= FALSE);
		mcMoveAbsX(
			Axis:= stAxisB, 
			Execute:= FALSE);
		nState := 58;				
	END_IF


58:
	ipMover.DisableExternalSetpointGeneration('disable ext. setpoints');
	nState := nState +1;
59:
	IF ipMover.P_DisableExternalSetpointGeneration.Done THEN
		nState := nState +1;
	END_IF
	
60:
	mcSetPos(
	Axis:= stAxisMaster , 
	Execute:= TRUE,
	Position := 0);
	IF mcSetPos.Done THEN
		mcSetPos(
			Axis:= stAxisMaster , 
			Execute:= FALSE);
		nstate := 70;
	END_IF
	
70:
	bExecute := FALSE;
	stReturn.Active := FALSE;
	streturn.Done := TRUE;
	nstate := 0;


	
	
END_CASE


CASE nstate OF
	20..60:
		
	
		ExtSetPos.x := stAxisX.NcToPlc.SetPos / 4.0; 
		ExtSetPos.y := stAxisY.NcToPlc.SetPos/ 4.0; 
		ExtSetPos.a := stAxisA.NcToPlc.SetPos * 20.0; 
		ExtSetPos.b := stAxisB.NcToPlc.SetPos* 20.0;	
	
		ExtSetVelo.x := stAxisX.NcToPlc.SetVelo/ 4.0; 
		ExtSetVelo.y := stAxisY.NcToPlc.SetVelo/ 4.0; 
		ExtSetVelo.a := stAxisA.NcToPlc.SetVelo* 20.0; 
		ExtSetVelo.b := stAxisB.NcToPlc.SetVelo* 20.0; 
	
		ExtSetAcc.x := stAxisX.NcToPlc.SetAcc/ 4.0; 
		ExtSetAcc.y := stAxisY.NcToPlc.SetAcc/ 4.0; 
		ExtSetAcc.a := stAxisA.NcToPlc.SetAcc* 20.0; 
		ExtSetAcc.b := stAxisB.NcToPlc.SetAcc* 20.0; 		
		
	
		ipMover.SetExternalSetpointValues(ExtSetPos,ExtSetVelo,ExtSetAcc);
END_CASE


IF mcMoveAbsMaster.Error THEN
	mcMoveAbsMaster(Axis := stAxisMaster,Execute := FALSE);
	nstate := -50;
END_IF

IF mcMoveAbsMaster.Error 
	OR mcMoveAbsA.error
	OR mcMoveAbsX.error
	OR mcPower.error
	OR mcSetPos.error
	OR McCamIn.error
	OR McCamOut.error THEN
	stReturn.Error := TRUE;
END_IF
END_METHOD

METHOD Cycle
VAR_INPUT
END_VAR
stAxisMaster.ReadStatus();
stAxisA.ReadStatus();
stAxisB.ReadStatus();
stAxisX.ReadStatus();
stAxisY.ReadStatus();

rtrigExecute(CLK:= bExecute, Q=> );
IF rtrigExecute.Q THEN
	MEMSET(destAddr:=ADR(stReturn) , fillByte:=0 , n:=SIZEOF(stReturn) );
END_IF


IF bExecute THEN
	ccl_StartMovement();
END_IF
END_METHOD

PROPERTY P_Return : REFERENCE to ST_CommandReturn
GET
P_Return ReF= stReturn;
END_GET
END_PROPERTY

METHOD StartMovement
VAR_INPUT
	NumCycles		: UINT;
	Velo			: LREAL;
END_VAR
nNumCycles := numCycles;
nVeloMaster := Velo;

bExecute := TRUE;
END_METHOD

END_FUNCTION_BLOCK

// ---- POUs/CustomerTemplates/GCode/FB_GCode.TcPOU
FUNCTION_BLOCK FB_GCode IMPLEMENTS I_GCode

VAR CONSTANT
	cNumItpAxes	: INT := 6;
END_VAR

VAR

// NC 

	mcPower			: MC_Power;

// G Code
	stItpAxis 				: ARRAY [1..6] OF AXIS_REF;
	stNciToPlc AT%I*		: NCTOPLC_NCICHANNEL_REF;
	stPlcToNci AT%Q*		: PLCTONC_NCICHANNEL_REF;
	fbCfgBuildExt3DGroup	: CfgBuildExt3DGroup;
	fbReconfigGroup			: CfgReconfigGroup;
	fbLoadProgram			: ItpLoadProgEx;
	fbStartStopProgram		: ItpStartStop;
	fbConfirmHandshake		: ItpConfirmHsk;
	fbItpReset				: ItpResetEx2;

	sGCodeFile				: STRING := 'C:\TwinCAT\Mc\Nci\EPBox.nc';
	
	fbGetBlockNum		: ItpGetBlockSearchData;
// ==	
	
	nState			: INT := 10;
	
	bStartCam		: BOOL;
	
	nAxesCnt		: INT := 1;
	ExtSetPos		: MoverVector;
	ExtSetVelo		: MoverVector;
	ExtSetAcc		: MoverVector;
	stExtSetPosOptions	: MC_EXTERNAL_SET_POSITION_MODE;	

	
	
// parameters

	
// internal
	bExecute		: BOOL;
	rtrigExecute 	: R_TRIG;
	stReturn		: ST_CommandReturn;
	
	bAllIptAxesEnabled	: BOOL;
	
	
END_VAR



VAR_IN_OUT
	ipMover			: I_XPlanarMoverStandard;
END_VAR

{attribute 'hide'}
METHOD PROTECTED ccl_StartMovement
VAR_INPUT
END_VAR
CASE nState OF

0:
 nstate := 10;

10:
	
	stExtSetPosOptions := MC_EXTERNAL_SET_POSITION_MODE.Relative;
	ipMover.EnableExternalSetpointGeneration('enable Ext Setpos',StExtSetPosOptions);	
	nState := 11;
11:
	IF ipMover.P_EnableExternalSetpointGeneration.Done  THEN
		nState := 14;
	END_IF		

14:

bAllIptAxesEnabled := TRUE;
FOR nAxesCnt := 1 TO cNumItpAxes DO
			mcPower(
				Axis:= stItpAxis[nAxesCnt], 
				Enable:= TRUE, 
				Enable_Positive:= TRUE, 
				Enable_Negative:= TRUE );
	
	bAllIptAxesEnabled := NOT stItpAxis[nAxesCnt].Status.Disabled AND bAllIptAxesEnabled;
END_FOR

IF bAllIptAxesEnabled THEN
	nstate := 15;
END_IF







	
15:

	Tc2_NCI.ItpSetOverridePercent(sPlcToNci:= stPlcToNci,fOverridePercent := 100);
	nState := 16;		
		
	16: 
		fbItpReset(sNciToPlc := stNciToPlc,
					bExecute := TRUE);

		IF NOT fbItpReset.bBusy THEN
			nState := 21;

			fbItpReset(sNciToPlc := stNciToPlc,
						bExecute := FALSE);
		END_IF	
		
	
	21: 
		fbCfgBuildExt3DGroup(
			bExecute:= TRUE, 
			nGroupId:= 6,
			nXAxisId:= 6 , 
			nYAxisId:= 7, 
			nZAxisId:= 0,
			bBusy=> , 
			bErr=> , 
			nErrId=> );

 
			IF NOT fbCfgBuildExt3DGroup.bBusy AND NOT fbCfgBuildExt3DGroup.bErr THEN
					fbCfgBuildExt3DGroup(
									bExecute:= FALSE);
				nState := 23;
			ELSIF fbCfgBuildExt3DGroup.bErr THEN
				nState := 999;
			END_IF	

	23: 
		fbLoadProgram( 
				sNciToPlc 	:= stNciToPlc,
				bExecute 	:= TRUE,
				sPrg		:= sGCodeFile,
				nLength		:= LEN(fbLoadProgram.sPrg));
		IF NOT fbLoadProgram.bBusy THEN
			fbLoadProgram( 
					sNciToPlc 	:= stNciToPlc,
					bExecute 	:= FALSE);
			nState := 24;
		END_IF	
		
	24:	
		fbStartStopProgram(nChnId := stNciToPlc.ChnId,
							bStart := TRUE,
							bStop := FALSE);
		
		IF NOT fbStartStopProgram.bBusy AND NOT fbStartStopProgram.bErr THEN
			fbStartStopProgram.bStart := FALSE;
			nState := 26;
		ELSIF fbStartStopProgram.bErr THEN
			fbStartStopProgram.bStart := FALSE;
			nState := 999;	
		END_IF


		

	26: // check handshake
	

		ExtSetPos.x := stItpAxis[1].NcToPlc.SetPos;
		ExtSetPos.y := stItpAxis[2].NcToPlc.SetPos;
		
		ExtSetVelo.x := stItpAxis[1].NcToPlc.SetVelo;
		ExtSetVelo.y := stItpAxis[2].NcToPlc.SetVelo;
		
		ExtSetAcc.x := stItpAxis[1].NcToPlc.SetAcc;
		ExtSetAcc.y := stItpAxis[2].NcToPlc.SetAcc;
		
		ipMover.SetExternalSetpointValues(ExtSetPos,ExtSetVelo,ExtSetAcc);
		
			
	
	
		IF ItpGetHskMFunc(sNciToPlc:=stNciToPlc) = 8 THEN
			nState := 30;
		END_IF

	
	
	30: 	
		fbConfirmHandshake( bExecute := TRUE,
							sNciToPlc := stNciToPlc,
							sPlcToNci := stPlcToNci);
							
		IF NOT fbConfirmHandshake.bBusy THEN
			fbConfirmHandshake( bExecute := FALSE,
								sNciToPlc := stNciToPlc,
								sPlcToNci := stPlcToNci);
			nState := 79;
		END_IF


79:

		fbStartStopProgram(nChnId := stNciToPlc.ChnId,
							bStart := FALSE,
							bStop := TRUE);

		
		 IF NOT fbStartStopProgram.bBusy THEN
				nState := 80;
		END_IF

80: fbReconfigGroup.bExecute := TRUE;
	nState := 81;
81:	
	
	IF NOT fbReconfigGroup.bBusy AND NOT fbReconfigGroup.bErr THEN
		fbReconfigGroup.bExecute := FALSE;
		nState := 90;
	ELSIF fbReconfigGroup.bErr THEN
		nState := 999;
		fbReconfigGroup.bExecute := FALSE;
	END_IF

90:
	ipMover.DisableExternalSetpointGeneration('');
	nstate := 91;
91:
	IF ipMover.P_DisableExternalSetpointGeneration.Done THEN
		nstate := 100;
	END_IF


	
100:
	stReturn.Done := TRUE;
	bExecute := FALSE;
	nState:= 0;	




END_CASE


CASE nstate OF
	20..90:
		
	
		ExtSetPos.x := stItpAxis[1] .NcToPlc.SetPos; 
		ExtSetPos.y := stItpAxis[2].NcToPlc.SetPos; 
		ExtSetPos.a := stItpAxis[4].NcToPlc.SetPos; 
		ExtSetPos.b := stItpAxis[5].NcToPlc.SetPos;	
	
		ExtSetVelo.x := stItpAxis[1].NcToPlc.SetVelo; 
		ExtSetVelo.y := stItpAxis[2].NcToPlc.SetVelo; 
		ExtSetVelo.a := stItpAxis[4].NcToPlc.SetVelo; 
		ExtSetVelo.b := stItpAxis[5].NcToPlc.SetVelo; 
	
		ExtSetAcc.x := stItpAxis[1].NcToPlc.SetAcc; 
		ExtSetAcc.y := stItpAxis[2].NcToPlc.SetAcc; 
		ExtSetAcc.a := stItpAxis[4].NcToPlc.SetAcc; 
		ExtSetAcc.b := stItpAxis[5].NcToPlc.SetAcc; 		
		
	
		ipMover.SetExternalSetpointValues(ExtSetPos,ExtSetVelo,ExtSetAcc);
END_CASE




IF fbLoadProgram.bErr
	OR fbStartStopProgram.bErr
	OR fbCfgBuildExt3DGroup.bErr
	OR fbReconfigGroup.bErr
	OR fbItpReset.bErr
	OR fbConfirmHandshake.bErr THEN
	stReturn.Error := TRUE;
END_IF
END_METHOD

METHOD Cycle
VAR
	nCnt	 : INT;
END_VAR
FOR nCnt := 1 TO cNumItpAxes DO
	stItpAxis[nCnt].ReadStatus();
END_FOR

rtrigExecute(CLK:= bExecute, Q=> );
IF rtrigExecute.Q THEN
	MEMSET(destAddr:=ADR(stReturn) , fillByte:=0 , n:=SIZEOF(stReturn) );
END_IF


IF bExecute THEN
	ccl_StartMovement();
END_IF
END_METHOD

PROPERTY P_Return : REFERENCE to ST_CommandReturn
GET
P_Return ReF= stReturn;
END_GET
END_PROPERTY

METHOD StartMovement
VAR_INPUT
	sFilePath	: STRING;
END_VAR


bExecute := TRUE;
END_METHOD

END_FUNCTION_BLOCK

// ---- POUs/FB_WriteLog.TcPOU
FUNCTION_BLOCK FB_WriteLog
VAR_INPUT
	sPath	: STRING;
	bErrorAcknowledge	: BOOL;
END_VAR
VAR_OUTPUT
END_VAR
VAR
	
	nState			: INT;
	hFile			: UINT;
	fbFileOpen		: FB_FileOpen;	
	fbFileWrite		: FB_FileWrite;
	fbFileClose		: FB_FileClose;	
	sWriteString	: STRING;
	fbFilePuts		: FB_FilePuts;
	
	sWriteLogArray 	: STRING;
	fbGetTime		: NT_GetTime;
	tTime			: TIME;
	nForCounter		: INT;
	stTimeZoneInfo	:  TC2_UTILITIES.ST_TimeZoneInformation;
	fbGetTimeZoneInformation: FB_GetTimeZoneInformation;
	

END_VAR
VAR CONSTANT
	nBufferSize : INT := 100;
END_VAR

	
CASE nState OF
	-1:
		
		IF bErrorAcknowledge THEN
			fbFileOpen(		bExecute	:= FALSE);
			bErrorAcknowledge := FALSE;
			nState := 0;
		END_IF



	0:	fbGetTimeZoneInformation(	sNetID 		:= '',
									bExecute 	:= TRUE,
									tzInfo		=> stTimeZoneInfo); 
		IF NOT fbGetTimeZoneInformation.bBusy THEN
			fbGetTimeZoneInformation(	sNetID 		:= '',
										bExecute 	:= FALSE);
			nState := 1;							
		END_IF							

	 	
	1:
			IF sWriteLogArray <> '' THEN
				
				sWriteString := sWriteLogArray;			
				FOR nForCounter:= 0 TO nBufferSize-1 DO
					sWriteLogArray[nForCounter]:= sWriteLogArray[nForCounter+1]; 	
				END_FOR
				nState := 5;
			END_IF
	
	5: fbFileOpen(
			sNetId		:='' , 
			sPathName	:=sPath , 
			nMode		:= FOPEN_MODEAPPEND, 
			ePath		:= PATH_GENERIC , 
			bExecute	:= TRUE, 
			tTimeout	:= , 
			bBusy		=> , 
			bError		=> , 
			nErrId		=> , 
			hFile		=>	hFile );
	
		IF NOT fbFileOpen.bBusy AND (fbFileOpen.hFile <> 0) THEN
			fbFileOpen(
			sNetId		:='' , 
			sPathName	:=sPath , 
			nMode		:= FOPEN_MODEAPPEND, 
			ePath		:= PATH_GENERIC , 
			bExecute	:= FALSE);
			nState := 10;
		ELSIF fbFileOpen.bError THEN
			nState := -1;
		END_IF 	
		
	10: 
	sWriteString := CONCAT(sWriteString,'$N');
		fbFilePuts(
			sNetId:='' , 
			hFile:=hFile , 
			sLine:=sWriteString , 
			bExecute:=TRUE , 
			tTimeout:= , 
			bBusy=> , 
			bError=> , 
			nErrId=> );
			
		IF NOT fbFilePuts.bBusy THEN
		
			fbFilePuts(
				sNetId:='' , 
				hFile:=hFile , 
				sLine:=sWriteString , 
				bExecute:=FALSE); 
			
			nState := 30;
		END_IF
		
	(*10: fbFileWrite(
			sNetId		:='' , 
			hFile		:= hFile , 
			pWriteBuff	:= ADR(sWriteString), 
			cbWriteLen	:= SIZEOF(sWriteString), 
			bExecute	:= TRUE, 
			tTimeout	:= , 
			bBusy		=> , 
			bError		=> , 
			nErrId		=> , 
			cbWrite		=> );
		
		IF NOT fbFileWrite.bBusy AND (fbFileWrite.cbWrite <> 0) THEN
			nState := 30;
			fbFileWrite(
			sNetId		:='' , 
			hFile		:= hFile , 
			bExecute	:= FALSE); 
		END_IF
		*)
	30: fbFileClose(
			sNetId:='' , 
			hFile:= hFile, 
			bExecute:= TRUE, 
			tTimeout:= , 
			bBusy=> , 
			bError=> , 
			nErrId=> );
			
		IF NOT fbFileClose.bBusy THEN
			 fbFileClose(
				sNetId:='' , 
				hFile:= hFile, 
				bExecute:= FALSE, 
				tTimeout:= , 
				bBusy=> , 
				bError=> , 
				nErrId=> );
				
				
				sWriteLogArray := '';
			nState := 0;
		END_IF

	
		
		

END_CASE

METHOD M_AddLogg
VAR_INPUT
	sParam : STRING;
END_VAR

VAR 
	lDCTime : ULINT;
	fbTimeConvert : FB_FileTimeToTzSpecificLocalTime; 

END_VAR

	IF sWriteLogArray = '' THEN
		
		lDCTime := F_GetActualDcTime64();
		fbTimeConvert(in:= DCTIME64_TO_FILETIME(lDcTime),tzInfo := stTimeZoneInfo);	
		
		sWriteLogArray := CONCAT(DCTIME64_TO_STRING(FILETIME_TO_DCTIME64(fbTimeConvert.out)),': ');
		sWriteLogArray := CONCAT(sWriteLogArray,sParam);
	END_IF
END_METHOD

END_FUNCTION_BLOCK

// ---- POUs/10_GeneralPlcBlocks/Blinker.TcPOU
PROGRAM Blinker
VAR
	
	fbBlinker1								:FB_Blinker;
	tTurnOffDelayB1							:TIME := T#1S;
	fbBlinker2								:FB_Blinker;
	
END_VAR
(* End *)

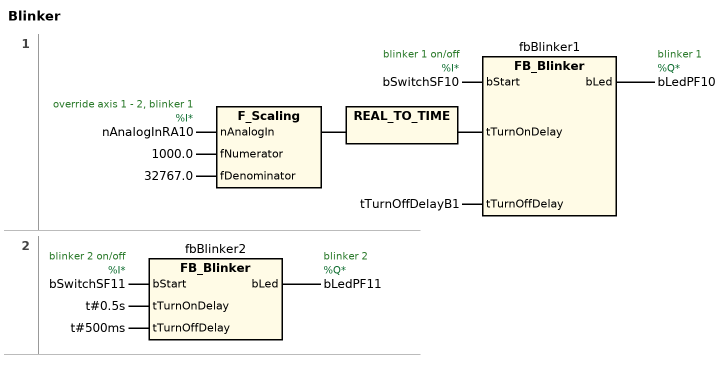
// NETWORK 1
//   bSwitchSF10: blinker 1 on/off | AT %I*
//   nAnalogInRA10: override axis 1 - 2, blinker 1 | AT %I*
//   bLedPF10: blinker 1 | AT %Q*
fbBlinker1(
    bStart := bSwitchSF10,
    tTurnOnDelay := REAL_TO_TIME(F_Scaling(nAnalogIn := nAnalogInRA10, fNumerator := 1000.0, fDenominator := 32767.0)),
    tTurnOffDelay := tTurnOffDelayB1); // FB_Blinker
bLedPF10 := fbBlinker1.bLed;

// NETWORK 2
//   bSwitchSF11: blinker 2 on/off | AT %I*
//   bLedPF11: blinker 2 | AT %Q*
fbBlinker2(bStart := bSwitchSF11, tTurnOnDelay := t#0.5s, tTurnOffDelay := t#500ms); // FB_Blinker
bLedPF11 := fbBlinker2.bLed;

END_PROGRAM

// ---- POUs/10_GeneralPlcBlocks/Components/F_Scaling.TcPOU
FUNCTION F_Scaling : REAL
VAR_INPUT

	nAnalogIn								:INT;
	fNumerator								:REAL;
	fDenominator							:REAL;
	
END_VAR
VAR
END_VAR
(* End *)

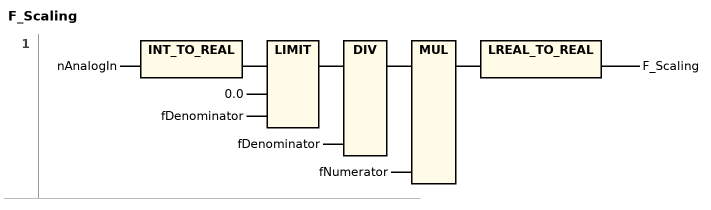
// NETWORK 1
F_Scaling := LREAL_TO_REAL((LIMIT(INT_TO_REAL(nAnalogIn), 0.0, fDenominator) / fDenominator) * fNumerator);

END_FUNCTION

// ---- POUs/10_GeneralPlcBlocks/ClockGenerator.TcPOU
PROGRAM ClockGenerator
VAR
	
	nCycleTime								:UDINT;		(* Cycle time from the PLC Task *)
	nTimeValue								:INT;		(* Time value clock generator*)
	
END_VAR
(* End *)

(* Clock generator *)

	(* PLC cycle time in ms  *)
	nCycleTime	:=	TwinCAT_SystemInfoVarList._TaskInfo[GETCURTASKINDEXEX()].cycleTime / 10000;

	(* Calculate with the cycle time the time value *)
	nTimeValue	:=	nTimeValue + UDINT_TO_INT(nCycleTime);

	(* Generate the clocks and the rising edges with the time value *)
	CASE nTimeValue OF

		500		:	bClock500ms			:=	TRUE;
					bRisingEdge500ms	:=	TRUE;

		1000	:	bClock500ms			:=	FALSE;
					bRisingEdge500ms	:=	TRUE;
					bClock1s			:=	TRUE;
					bRisingEdge1s		:=	TRUE;

		1500	:	bClock500ms			:=	TRUE;
					bRisingEdge500ms	:=	TRUE;

		2000	:	bClock500ms			:=	FALSE;
					bRisingEdge500ms	:=	TRUE;
					bClock1s			:=	FALSE;
					bRisingEdge1s		:=	TRUE;
					bClock2s			:=	TRUE;
					bRisingEdge2s		:=	TRUE;

		2500	:	bClock500ms			:=	TRUE;
					bRisingEdge500ms	:=	TRUE;

		3000	:	bClock500ms			:=	FALSE;
					bRisingEdge500ms	:=	TRUE;
					bClock1s			:=	TRUE;
					bRisingEdge1s		:=	TRUE;

		3500	:	bClock500ms			:=	TRUE;
					bRisingEdge500ms	:=	TRUE;

		4000	:	bClock500ms			:=	FALSE;
					bRisingEdge500ms	:=	TRUE;
			 		bClock1s			:=	FALSE;
					bRisingEdge1s		:=	TRUE;
					bClock2s			:=	FALSE;
					bRisingEdge2s		:=	TRUE;
					
	ELSE

		(* Reset the rising edge variables after one cycle *)
		bRisingEdge500ms	:=	FALSE;
		bRisingEdge1s		:=	FALSE;
		bRisingEdge2s		:=	FALSE;

	END_CASE;

	(* Sequence reset at 4000ms *)
	IF nTimeValue >= 4000
	THEN
		nTimeValue := 0;
	END_IF

(* End *)

END_PROGRAM

// ---- POUs/10_GeneralPlcBlocks/GeneralPlc.TcPOU
PROGRAM GeneralPlc
VAR
END_VAR
(* End *)

(* General *)

(* Led on/off *)

	bLedPF14 := bSwitchSF14;
	
	bLedPF15 := bSwitchSF15;
	
	bLedPF22 := bSwitchSF22;
	
	bLedPF25 := bSwitchSF25;

(* End *)

END_PROGRAM
